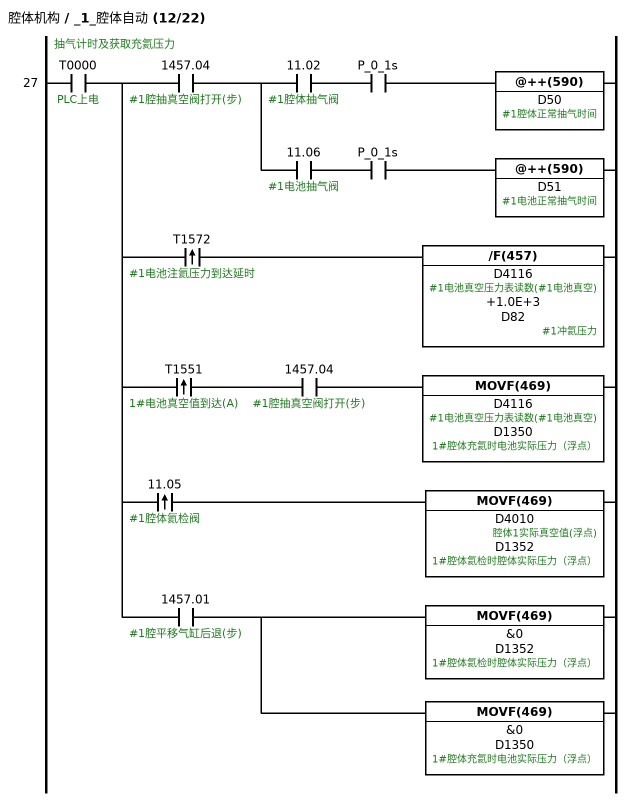
; [picture p288: 腔体机构 / _1_腔体自动, rungs 27-27]
; rung 27: 抽气计时及获取充氦压力
LD T0000  ; PLC上电
OUT TR0
AND 1457.04  ; #1腔抽真空阀打开(步)
OUT TR1
AND 11.02  ; #1腔体抽气阀
AND P_0_1s
@++(590) D50  ; #1腔体正常抽气时间
LD TR1
AND 11.06  ; #1电池抽气阀
AND P_0_1s
@++(590) D51  ; #1电池正常抽气时间
LD TR0
@AND T1572  ; #1电池注氦压力到达延时
/F(457) D4116 +1.0E+3 D82  ; #1电池真空压力表读数(#1电池真空), #1冲氦压力
LD TR0
@AND T1551  ; 1#电池真空值到达(A)
AND 1457.04  ; #1腔抽真空阀打开(步)
MOVF(469) D4116 D1350  ; #1电池真空压力表读数(#1电池真空), 1#腔体充氦时电池实际压力（浮点）
LD TR0
@AND 11.05  ; #1腔体氦检阀
MOVF(469) D4010 D1352  ; 腔体1实际真空值(浮点), 1#腔体氦检时腔体实际压力（浮点）
LD TR0
AND 1457.01  ; #1腔平移气缸后退(步)
MOVF(469) &0 D1352  ; 1#腔体氦检时腔体实际压力（浮点）
MOVF(469) &0 D1350  ; 1#腔体充氦时电池实际压力（浮点）

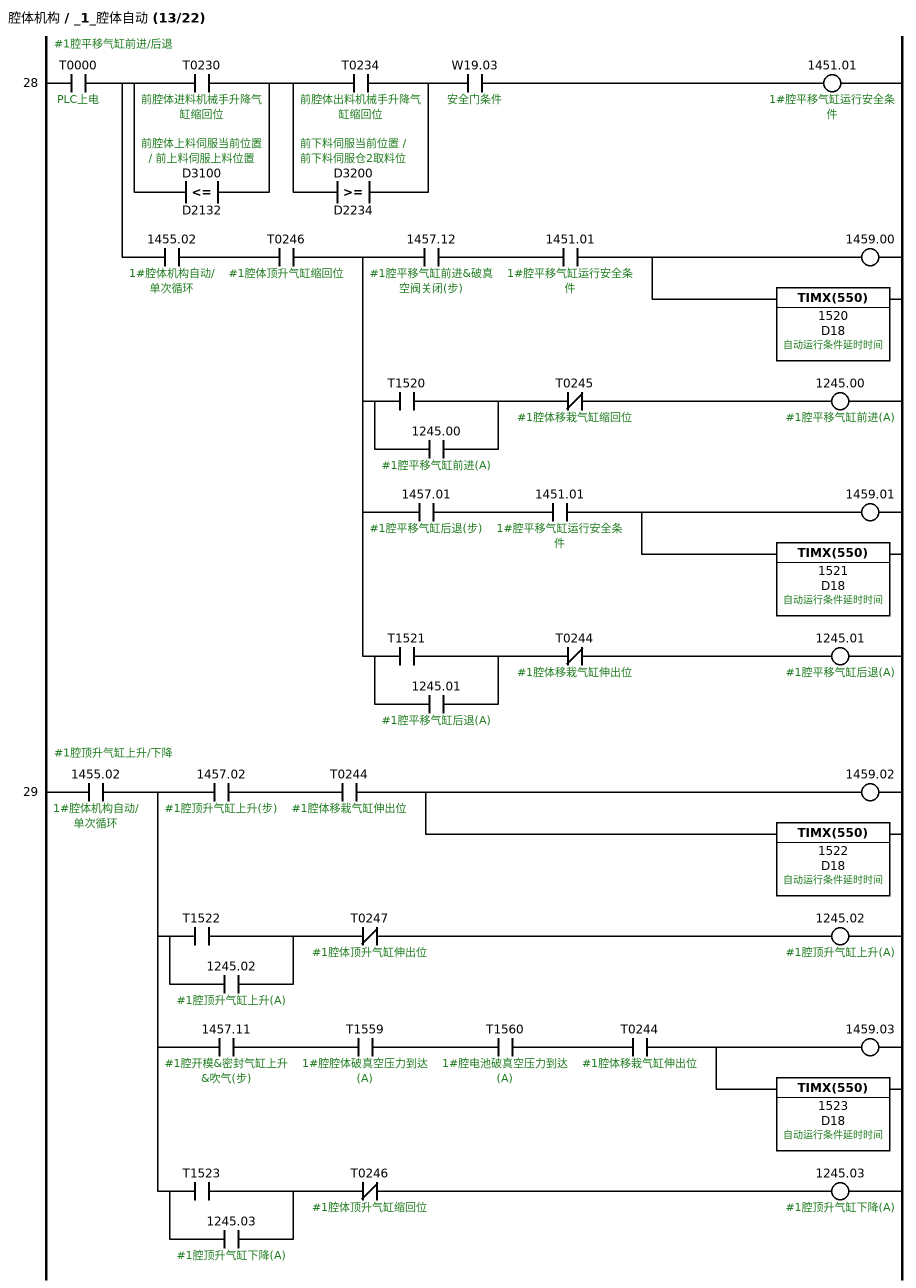
; rung 28: #1腔平移气缸前进/后退
LD T0000  ; PLC上电
OUT TR0
LD T0230  ; 前腔体进料机械手升降气缸缩回位
OR<=SL(318) D3100 D2132  ; 前腔体上料伺服当前位置, 前上料伺服上料位置
ANDLD
LD T0234  ; 前腔体出料机械手升降气缸缩回位
OR>=SL(328) D3200 D2234  ; 前下料伺服当前位置, 前下料伺服仓2取料位
ANDLD
AND W19.03  ; 安全门条件
OUT 1451.01  ; 1#腔平移气缸运行安全条件
LD TR0
AND 1455.02  ; 1#腔体机构自动/单次循环
AND T0246  ; #1腔体顶升气缸缩回位
OUT TR0
AND 1457.12  ; #1腔平移气缸前进&破真空阀关闭(步)
AND 1451.01  ; 1#腔平移气缸运行安全条件
OUT 1459.00
TIMX(550) 1520 D18  ; 自动运行条件延时时间
LD TR0
LD T1520
OR 1245.00  ; #1腔平移气缸前进(A)
ANDLD
ANDNOT T0245  ; #1腔体移栽气缸缩回位
OUT 1245.00  ; #1腔平移气缸前进(A)
LD TR0
AND 1457.01  ; #1腔平移气缸后退(步)
AND 1451.01  ; 1#腔平移气缸运行安全条件
OUT 1459.01
TIMX(550) 1521 D18  ; 自动运行条件延时时间
LD TR0
LD T1521
OR 1245.01  ; #1腔平移气缸后退(A)
ANDLD
ANDNOT T0244  ; #1腔体移栽气缸伸出位
OUT 1245.01  ; #1腔平移气缸后退(A)
; rung 29: #1腔顶升气缸上升/下降
LD 1455.02  ; 1#腔体机构自动/单次循环
OUT TR0
AND 1457.02  ; #1腔顶升气缸上升(步)
AND T0244  ; #1腔体移栽气缸伸出位
OUT 1459.02
TIMX(550) 1522 D18  ; 自动运行条件延时时间
LD TR0
LD T1522
OR 1245.02  ; #1腔顶升气缸上升(A)
ANDLD
ANDNOT T0247  ; #1腔体顶升气缸伸出位
OUT 1245.02  ; #1腔顶升气缸上升(A)
LD TR0
AND 1457.11  ; #1腔开模&密封气缸上升&吹气(步)
AND T1559  ; 1#腔腔体破真空压力到达(A)
AND T1560  ; 1#腔电池破真空压力到达(A)
AND T0244  ; #1腔体移栽气缸伸出位
OUT 1459.03
TIMX(550) 1523 D18  ; 自动运行条件延时时间
LD TR0
LD T1523
OR 1245.03  ; #1腔顶升气缸下降(A)
ANDLD
ANDNOT T0246  ; #1腔体顶升气缸缩回位
OUT 1245.03  ; #1腔顶升气缸下降(A)

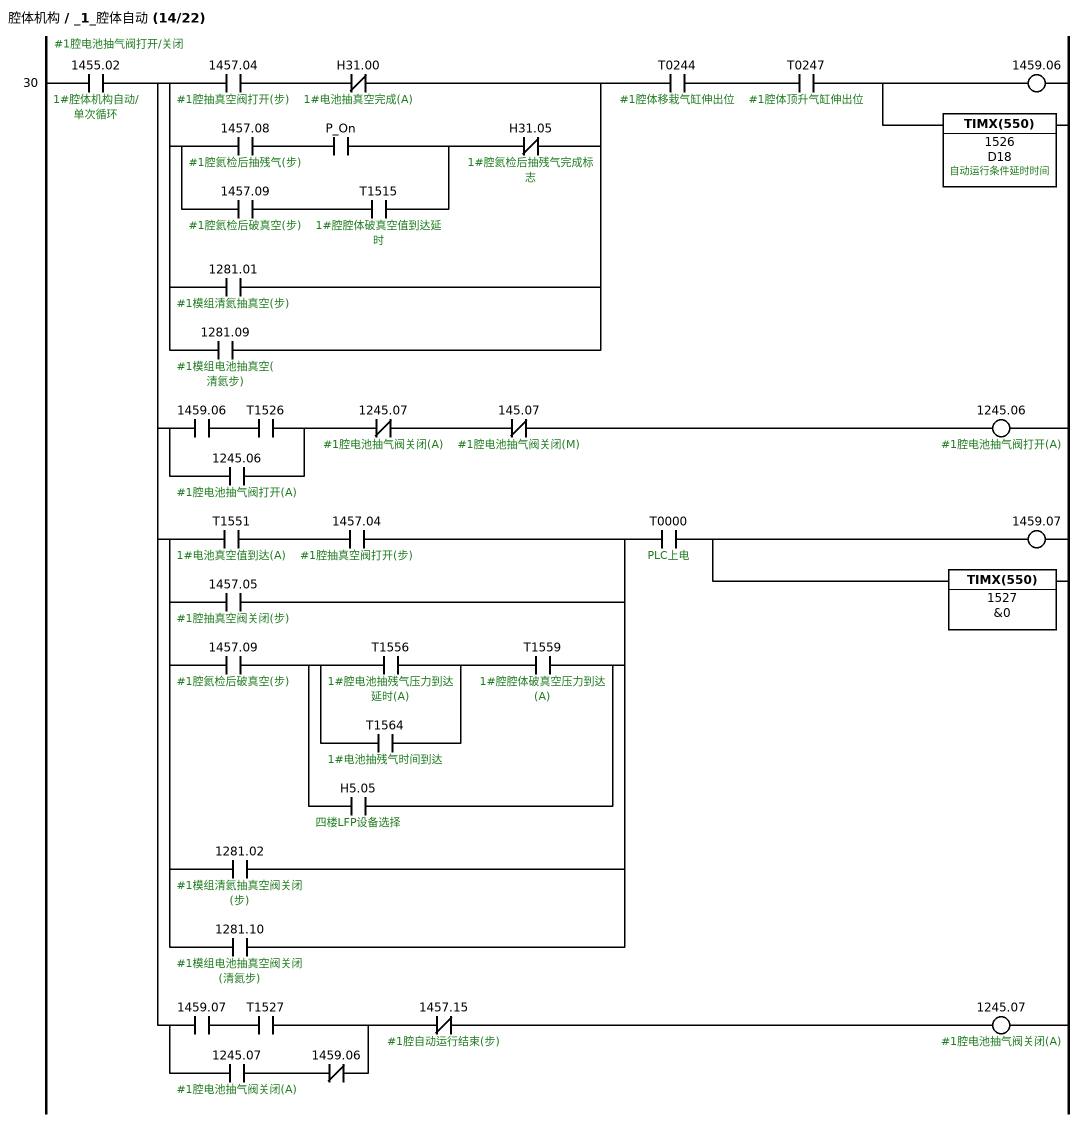
; rung 30: #1腔电池抽气阀打开/关闭
LD 1455.02  ; 1#腔体机构自动/单次循环
OUT TR0
LD 1457.04  ; #1腔抽真空阀打开(步)
ANDNOT H31.00  ; 1#电池抽真空完成(A)
LD 1457.08  ; #1腔氦检后抽残气(步)
AND P_On
LD 1457.09  ; #1腔氦检后破真空(步)
AND T1515  ; 1#腔腔体破真空值到达延时
ORLD
ANDNOT H31.05  ; 1#腔氦检后抽残气完成标志
ORLD
OR 1281.01  ; #1模组清氦抽真空(步)
OR 1281.09  ; #1模组电池抽真空(清氦步)
ANDLD
AND T0244  ; #1腔体移栽气缸伸出位
AND T0247  ; #1腔体顶升气缸伸出位
OUT 1459.06
TIMX(550) 1526 D18  ; 自动运行条件延时时间
LD TR0
LD 1459.06
AND T1526
OR 1245.06  ; #1腔电池抽气阀打开(A)
ANDLD
ANDNOT 1245.07  ; #1腔电池抽气阀关闭(A)
ANDNOT 145.07  ; #1腔电池抽气阀关闭(M)
OUT 1245.06  ; #1腔电池抽气阀打开(A)
LD TR0
LD T1551  ; 1#电池真空值到达(A)
AND 1457.04  ; #1腔抽真空阀打开(步)
OR 1457.05  ; #1腔抽真空阀关闭(步)
LD 1457.09  ; #1腔氦检后破真空(步)
LD T1556  ; 1#腔电池抽残气压力到达延时(A)
OR T1564  ; 1#电池抽残气时间到达
AND T1559  ; 1#腔腔体破真空压力到达(A)
OR H5.05  ; 四楼LFP设备选择
ANDLD
ORLD
OR 1281.02  ; #1模组清氦抽真空阀关闭(步)
OR 1281.10  ; #1模组电池抽真空阀关闭(清氦步)
ANDLD
AND T0000  ; PLC上电
OUT 1459.07
TIMX(550) 1527 &0
LD TR0
LD 1459.07
AND T1527
LD 1245.07  ; #1腔电池抽气阀关闭(A)
ANDNOT 1459.06
ORLD
ANDLD
ANDNOT 1457.15  ; #1腔自动运行结束(步)
OUT 1245.07  ; #1腔电池抽气阀关闭(A)

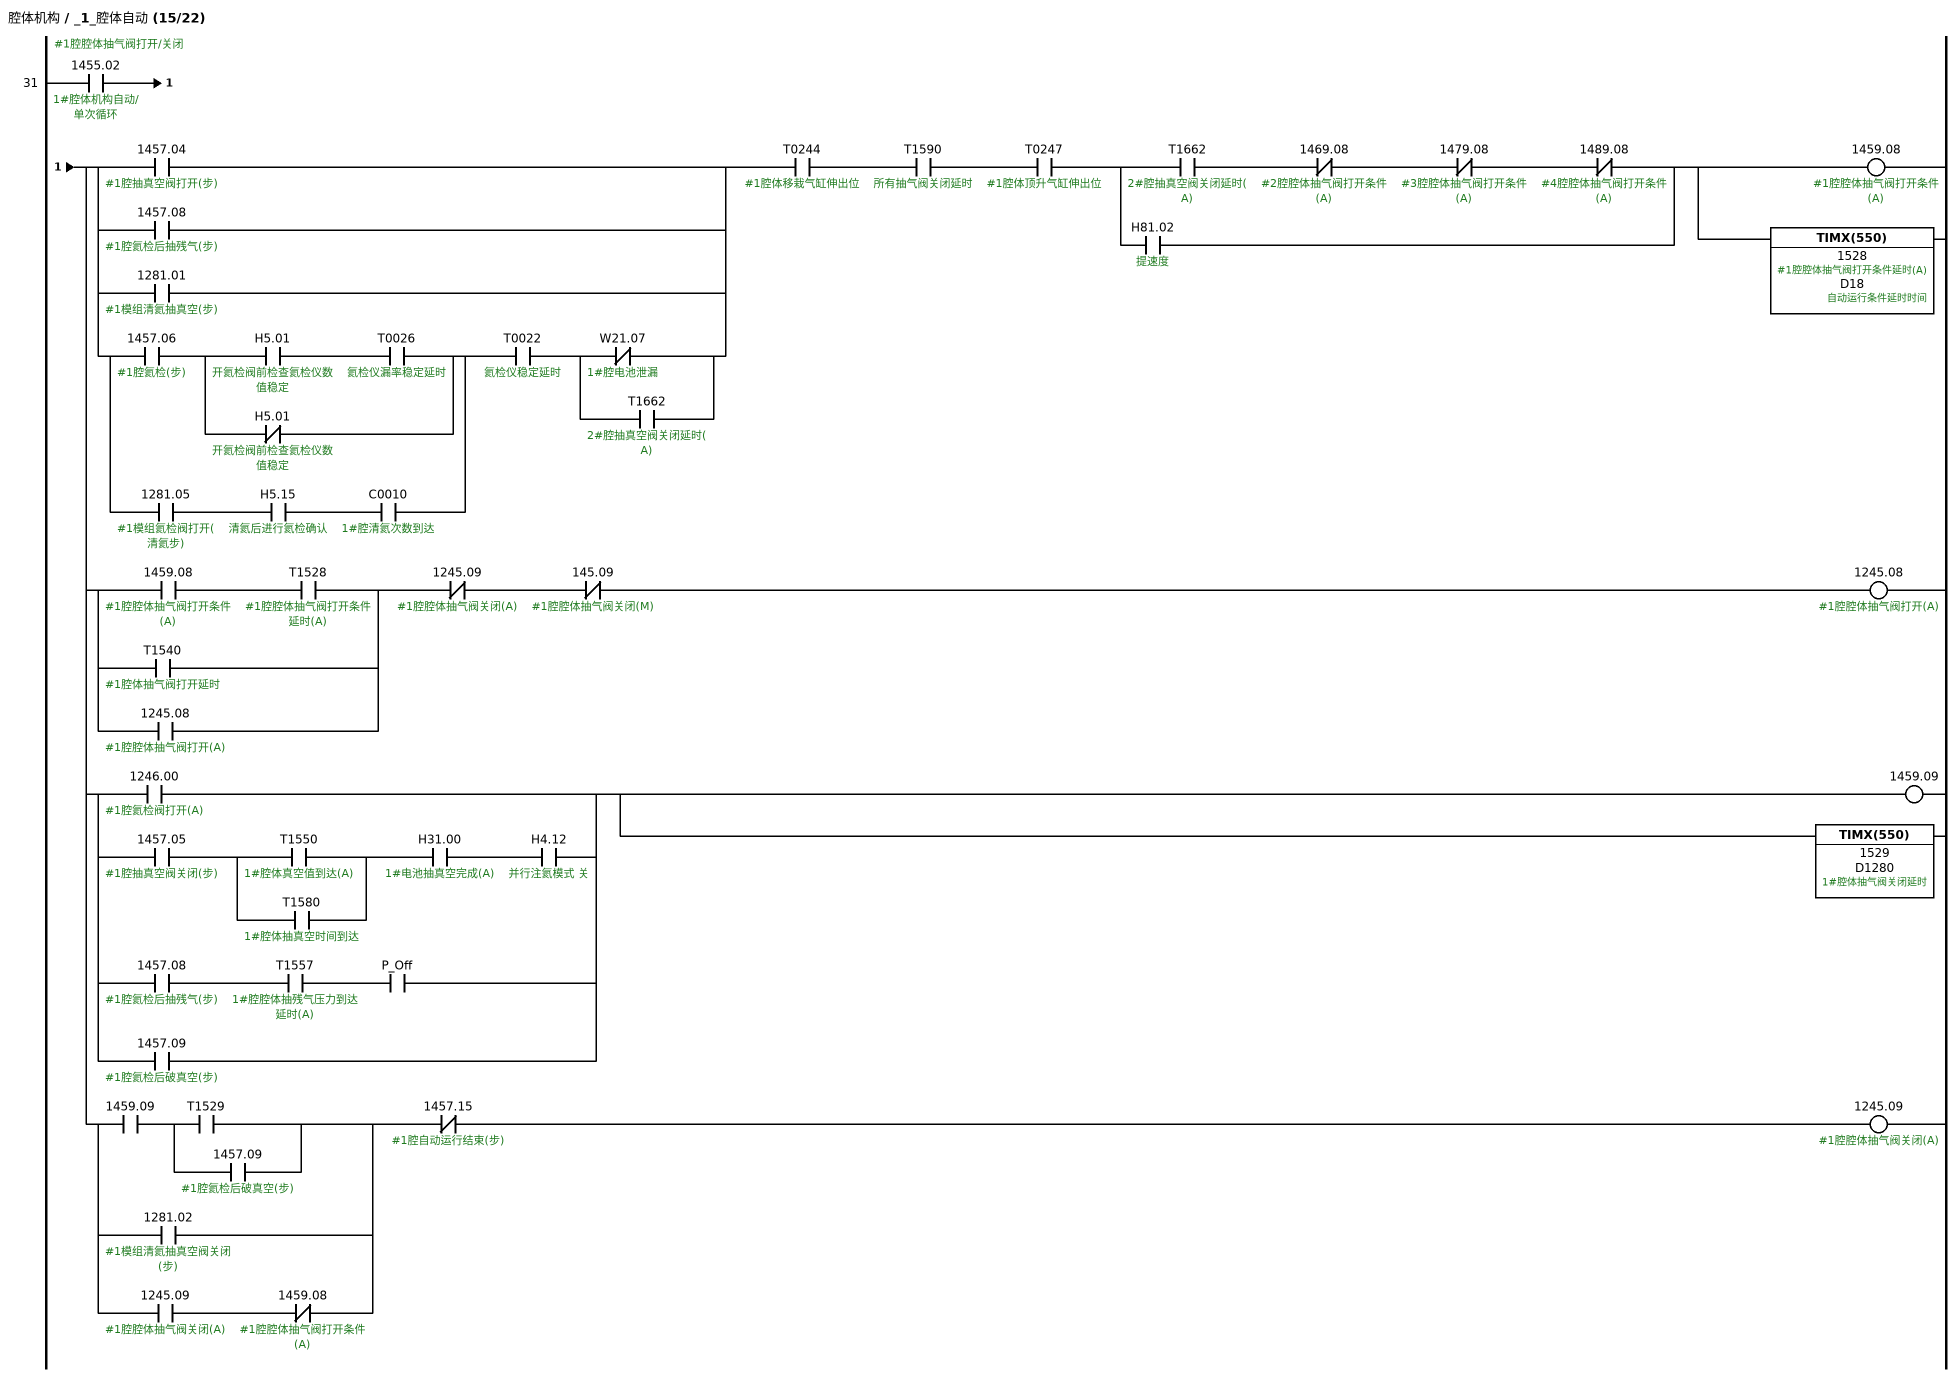
; rung 31: #1腔腔体抽气阀打开/关闭
LD 1455.02  ; 1#腔体机构自动/单次循环
OUT TR0
LD 1457.04  ; #1腔抽真空阀打开(步)
OR 1457.08  ; #1腔氦检后抽残气(步)
OR 1281.01  ; #1模组清氦抽真空(步)
LD 1457.06  ; #1腔氦检(步)
LD H5.01  ; 开氦检阀前检查氦检仪数值稳定
AND T0026  ; 氦检仪漏率稳定延时
ORNOT H5.01  ; 开氦检阀前检查氦检仪数值稳定
ANDLD
LD 1281.05  ; #1模组氦检阀打开(清氦步)
AND H5.15  ; 清氦后进行氦检确认
AND C0010  ; 1#腔清氦次数到达
ORLD
AND T0022  ; 氦检仪稳定延时
LDNOT W21.07  ; 1#腔电池泄漏
OR T1662  ; 2#腔抽真空阀关闭延时(A)
ANDLD
ORLD
ANDLD
AND T0244  ; #1腔体移栽气缸伸出位
AND T1590  ; 所有抽气阀关闭延时
AND T0247  ; #1腔体顶升气缸伸出位
LD T1662  ; 2#腔抽真空阀关闭延时(A)
ANDNOT 1469.08  ; #2腔腔体抽气阀打开条件(A)
ANDNOT 1479.08  ; #3腔腔体抽气阀打开条件(A)
ANDNOT 1489.08  ; #4腔腔体抽气阀打开条件(A)
OR H81.02  ; 提速度
ANDLD
OUT 1459.08  ; #1腔腔体抽气阀打开条件(A)
TIMX(550) 1528 D18  ; 自动运行条件延时时间, #1腔腔体抽气阀打开条件延时(A)
LD TR0
LD 1459.08  ; #1腔腔体抽气阀打开条件(A)
AND T1528  ; #1腔腔体抽气阀打开条件延时(A)
OR T1540  ; #1腔体抽气阀打开延时
OR 1245.08  ; #1腔腔体抽气阀打开(A)
ANDLD
ANDNOT 1245.09  ; #1腔腔体抽气阀关闭(A)
ANDNOT 145.09  ; #1腔腔体抽气阀关闭(M)
OUT 1245.08  ; #1腔腔体抽气阀打开(A)
LD TR0
LD 1246.00  ; #1腔氦检阀打开(A)
LD 1457.05  ; #1腔抽真空阀关闭(步)
LD T1550  ; 1#腔体真空值到达(A)
OR T1580  ; 1#腔体抽真空时间到达
ANDLD
AND H31.00  ; 1#电池抽真空完成(A)
AND H4.12  ; 并行注氦模式 关
ORLD
LD 1457.08  ; #1腔氦检后抽残气(步)
AND T1557  ; 1#腔腔体抽残气压力到达延时(A)
AND P_Off
ORLD
OR 1457.09  ; #1腔氦检后破真空(步)
ANDLD
OUT 1459.09
TIMX(550) 1529 D1280  ; 1#腔体抽气阀关闭延时
LD TR0
LD 1459.09
LD T1529
OR 1457.09  ; #1腔氦检后破真空(步)
ANDLD
OR 1281.02  ; #1模组清氦抽真空阀关闭(步)
LD 1245.09  ; #1腔腔体抽气阀关闭(A)
ANDNOT 1459.08  ; #1腔腔体抽气阀打开条件(A)
ORLD
ANDLD
ANDNOT 1457.15  ; #1腔自动运行结束(步)
OUT 1245.09  ; #1腔腔体抽气阀关闭(A)

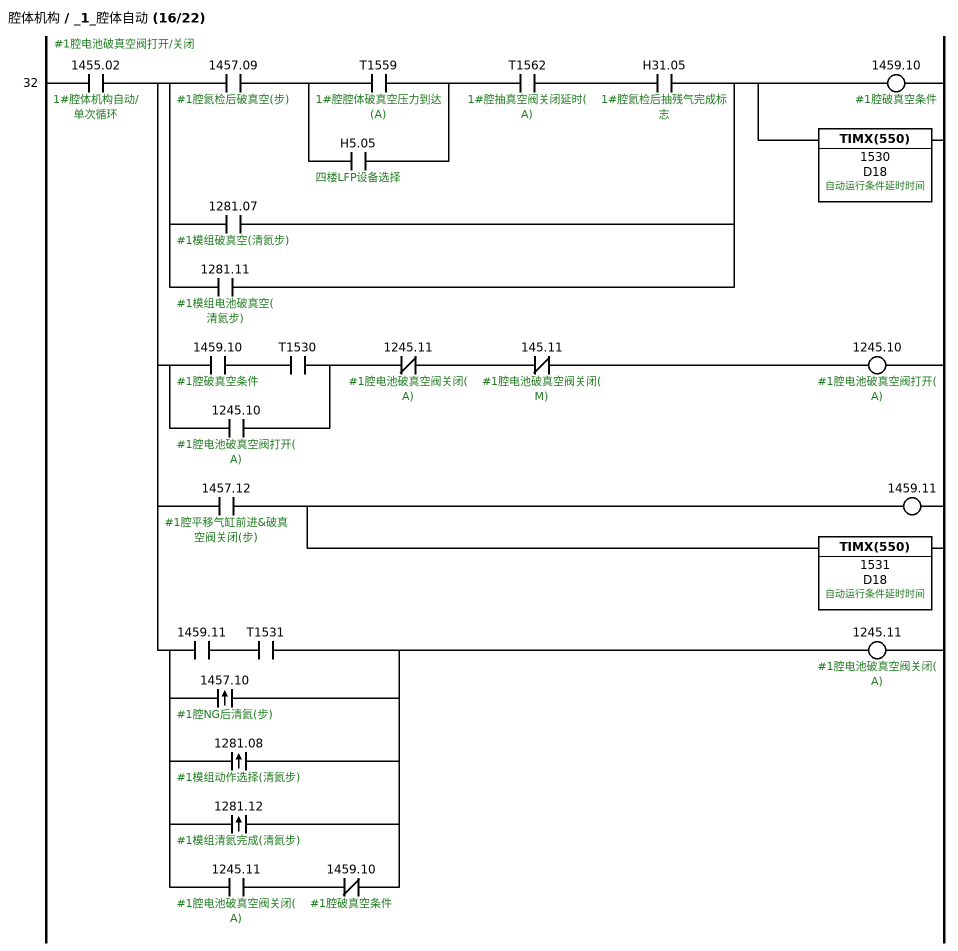
; rung 32: #1腔电池破真空阀打开/关闭
LD 1455.02  ; 1#腔体机构自动/单次循环
OUT TR0
LD 1457.09  ; #1腔氦检后破真空(步)
LD T1559  ; 1#腔腔体破真空压力到达(A)
OR H5.05  ; 四楼LFP设备选择
ANDLD
AND T1562  ; 1#腔抽真空阀关闭延时(A)
AND H31.05  ; 1#腔氦检后抽残气完成标志
OR 1281.07  ; #1模组破真空(清氦步)
OR 1281.11  ; #1模组电池破真空(清氦步)
ANDLD
OUT 1459.10  ; #1腔破真空条件
TIMX(550) 1530 D18  ; 自动运行条件延时时间
LD TR0
LD 1459.10  ; #1腔破真空条件
AND T1530
OR 1245.10  ; #1腔电池破真空阀打开(A)
ANDLD
ANDNOT 1245.11  ; #1腔电池破真空阀关闭(A)
ANDNOT 145.11  ; #1腔电池破真空阀关闭(M)
OUT 1245.10  ; #1腔电池破真空阀打开(A)
LD TR0
AND 1457.12  ; #1腔平移气缸前进&破真空阀关闭(步)
OUT 1459.11
TIMX(550) 1531 D18  ; 自动运行条件延时时间
LD TR0
LD 1459.11
AND T1531
@OR 1457.10  ; #1腔NG后清氦(步)
@OR 1281.08  ; #1模组动作选择(清氦步)
@OR 1281.12  ; #1模组清氦完成(清氦步)
LD 1245.11  ; #1腔电池破真空阀关闭(A)
ANDNOT 1459.10  ; #1腔破真空条件
ORLD
ANDLD
OUT 1245.11  ; #1腔电池破真空阀关闭(A)

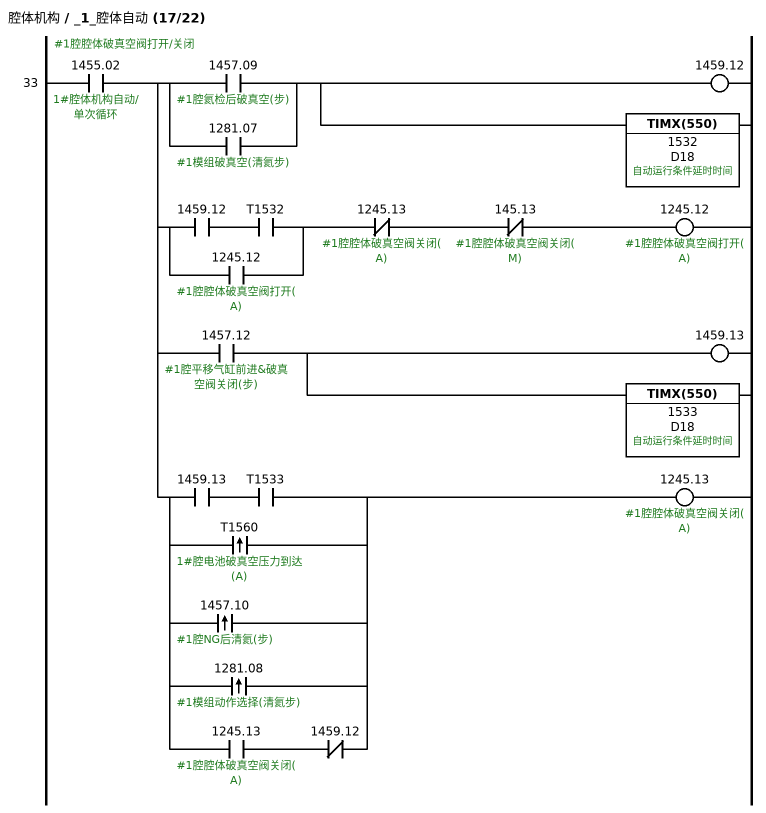
; rung 33: #1腔腔体破真空阀打开/关闭
LD 1455.02  ; 1#腔体机构自动/单次循环
OUT TR0
LD 1457.09  ; #1腔氦检后破真空(步)
OR 1281.07  ; #1模组破真空(清氦步)
ANDLD
OUT 1459.12
TIMX(550) 1532 D18  ; 自动运行条件延时时间
LD TR0
LD 1459.12
AND T1532
OR 1245.12  ; #1腔腔体破真空阀打开(A)
ANDLD
ANDNOT 1245.13  ; #1腔腔体破真空阀关闭(A)
ANDNOT 145.13  ; #1腔腔体破真空阀关闭(M)
OUT 1245.12  ; #1腔腔体破真空阀打开(A)
LD TR0
AND 1457.12  ; #1腔平移气缸前进&破真空阀关闭(步)
OUT 1459.13
TIMX(550) 1533 D18  ; 自动运行条件延时时间
LD TR0
LD 1459.13
AND T1533
@OR T1560  ; 1#腔电池破真空压力到达(A)
@OR 1457.10  ; #1腔NG后清氦(步)
@OR 1281.08  ; #1模组动作选择(清氦步)
LD 1245.13  ; #1腔腔体破真空阀关闭(A)
ANDNOT 1459.12
ORLD
ANDLD
OUT 1245.13  ; #1腔腔体破真空阀关闭(A)

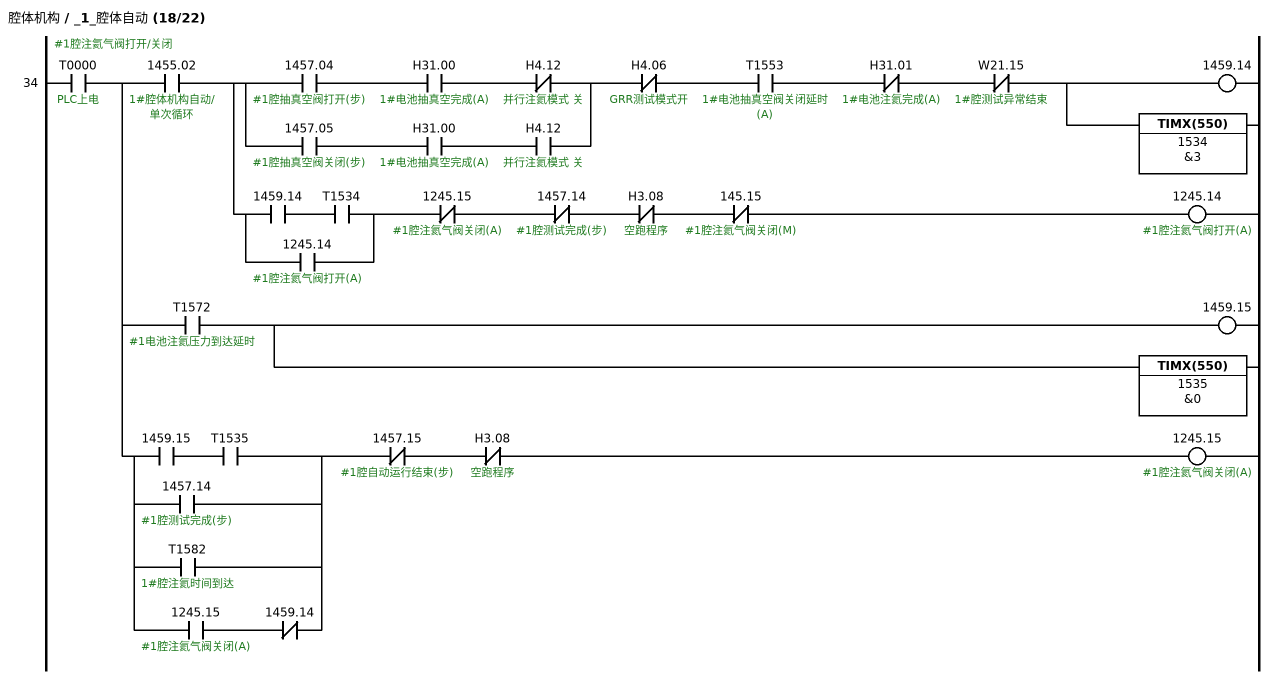
; rung 34: #1腔注氦气阀打开/关闭
LD T0000  ; PLC上电
OUT TR0
AND 1455.02  ; 1#腔体机构自动/单次循环
OUT TR1
LD 1457.04  ; #1腔抽真空阀打开(步)
AND H31.00  ; 1#电池抽真空完成(A)
ANDNOT H4.12  ; 并行注氦模式 关
LD 1457.05  ; #1腔抽真空阀关闭(步)
AND H31.00  ; 1#电池抽真空完成(A)
AND H4.12  ; 并行注氦模式 关
ORLD
ANDLD
ANDNOT H4.06  ; GRR测试模式开
AND T1553  ; 1#电池抽真空阀关闭延时(A)
ANDNOT H31.01  ; 1#电池注氦完成(A)
ANDNOT W21.15  ; 1#腔测试异常结束
OUT 1459.14
TIMX(550) 1534 &3
LD TR1
LD 1459.14
AND T1534
OR 1245.14  ; #1腔注氦气阀打开(A)
ANDLD
ANDNOT 1245.15  ; #1腔注氦气阀关闭(A)
ANDNOT 1457.14  ; #1腔测试完成(步)
ANDNOT H3.08  ; 空跑程序
ANDNOT 145.15  ; #1腔注氦气阀关闭(M)
OUT 1245.14  ; #1腔注氦气阀打开(A)
LD TR0
AND T1572  ; #1电池注氦压力到达延时
OUT 1459.15
TIMX(550) 1535 &0
LD TR0
LD 1459.15
AND T1535
OR 1457.14  ; #1腔测试完成(步)
OR T1582  ; 1#腔注氦时间到达
LD 1245.15  ; #1腔注氦气阀关闭(A)
ANDNOT 1459.14
ORLD
ANDLD
ANDNOT 1457.15  ; #1腔自动运行结束(步)
ANDNOT H3.08  ; 空跑程序
OUT 1245.15  ; #1腔注氦气阀关闭(A)

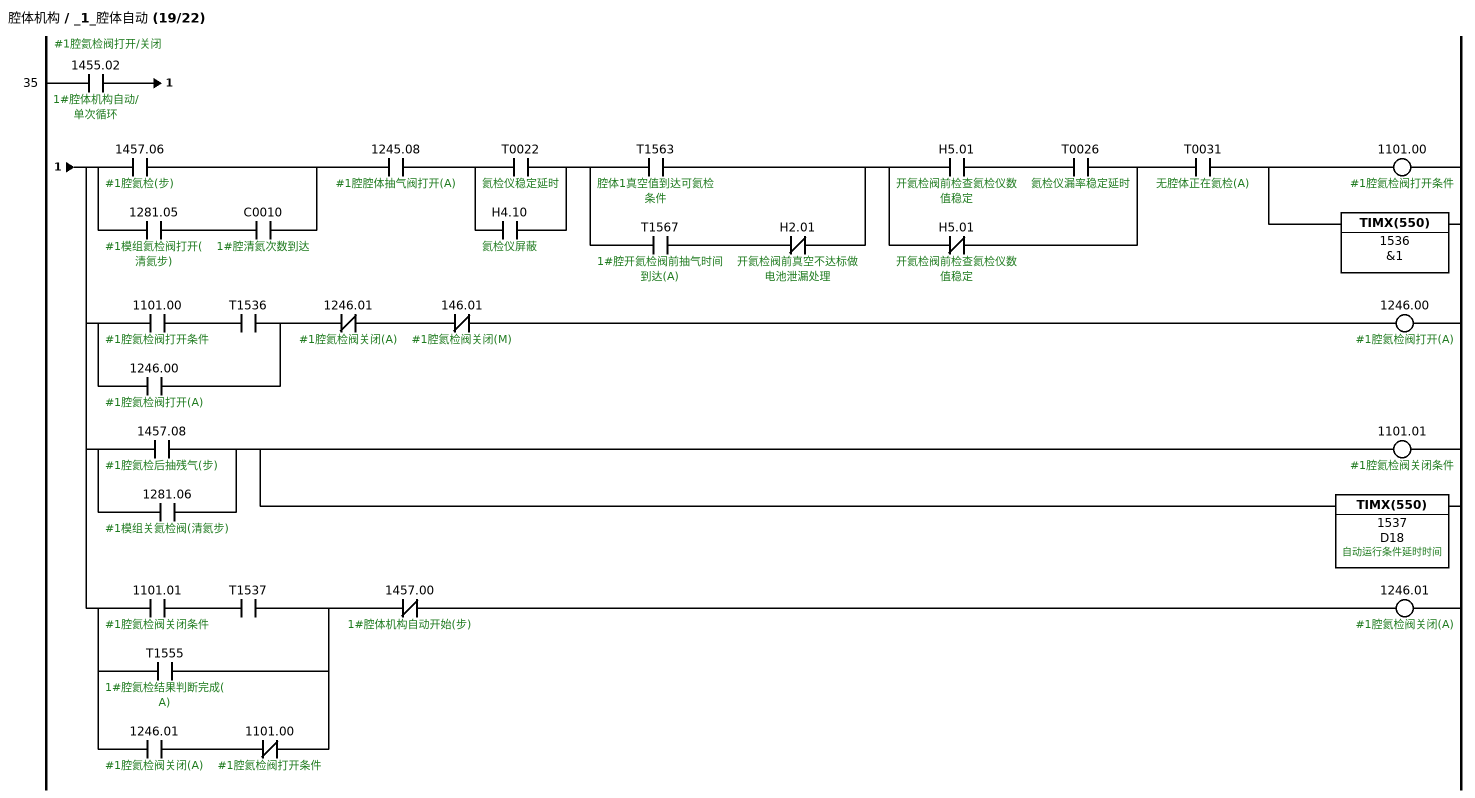
; rung 35: #1腔氦检阀打开/关闭
LD 1455.02  ; 1#腔体机构自动/单次循环
OUT TR0
LD 1457.06  ; #1腔氦检(步)
LD 1281.05  ; #1模组氦检阀打开(清氦步)
AND C0010  ; 1#腔清氦次数到达
ORLD
ANDLD
AND 1245.08  ; #1腔腔体抽气阀打开(A)
LD T0022  ; 氦检仪稳定延时
OR H4.10  ; 氦检仪屏蔽
ANDLD
LD T1563  ; 腔体1真空值到达可氦检条件
LD T1567  ; 1#腔开氦检阀前抽气时间到达(A)
ANDNOT H2.01  ; 开氦检阀前真空不达标做电池泄漏处理
ORLD
ANDLD
LD H5.01  ; 开氦检阀前检查氦检仪数值稳定
AND T0026  ; 氦检仪漏率稳定延时
ORNOT H5.01  ; 开氦检阀前检查氦检仪数值稳定
ANDLD
AND T0031  ; 无腔体正在氦检(A)
OUT 1101.00  ; #1腔氦检阀打开条件
TIMX(550) 1536 &1
LD TR0
LD 1101.00  ; #1腔氦检阀打开条件
AND T1536
OR 1246.00  ; #1腔氦检阀打开(A)
ANDLD
ANDNOT 1246.01  ; #1腔氦检阀关闭(A)
ANDNOT 146.01  ; #1腔氦检阀关闭(M)
OUT 1246.00  ; #1腔氦检阀打开(A)
LD TR0
LD 1457.08  ; #1腔氦检后抽残气(步)
OR 1281.06  ; #1模组关氦检阀(清氦步)
ANDLD
OUT 1101.01  ; #1腔氦检阀关闭条件
TIMX(550) 1537 D18  ; 自动运行条件延时时间
LD TR0
LD 1101.01  ; #1腔氦检阀关闭条件
AND T1537
OR T1555  ; 1#腔氦检结果判断完成(A)
LD 1246.01  ; #1腔氦检阀关闭(A)
ANDNOT 1101.00  ; #1腔氦检阀打开条件
ORLD
ANDLD
ANDNOT 1457.00  ; 1#腔体机构自动开始(步)
OUT 1246.01  ; #1腔氦检阀关闭(A)

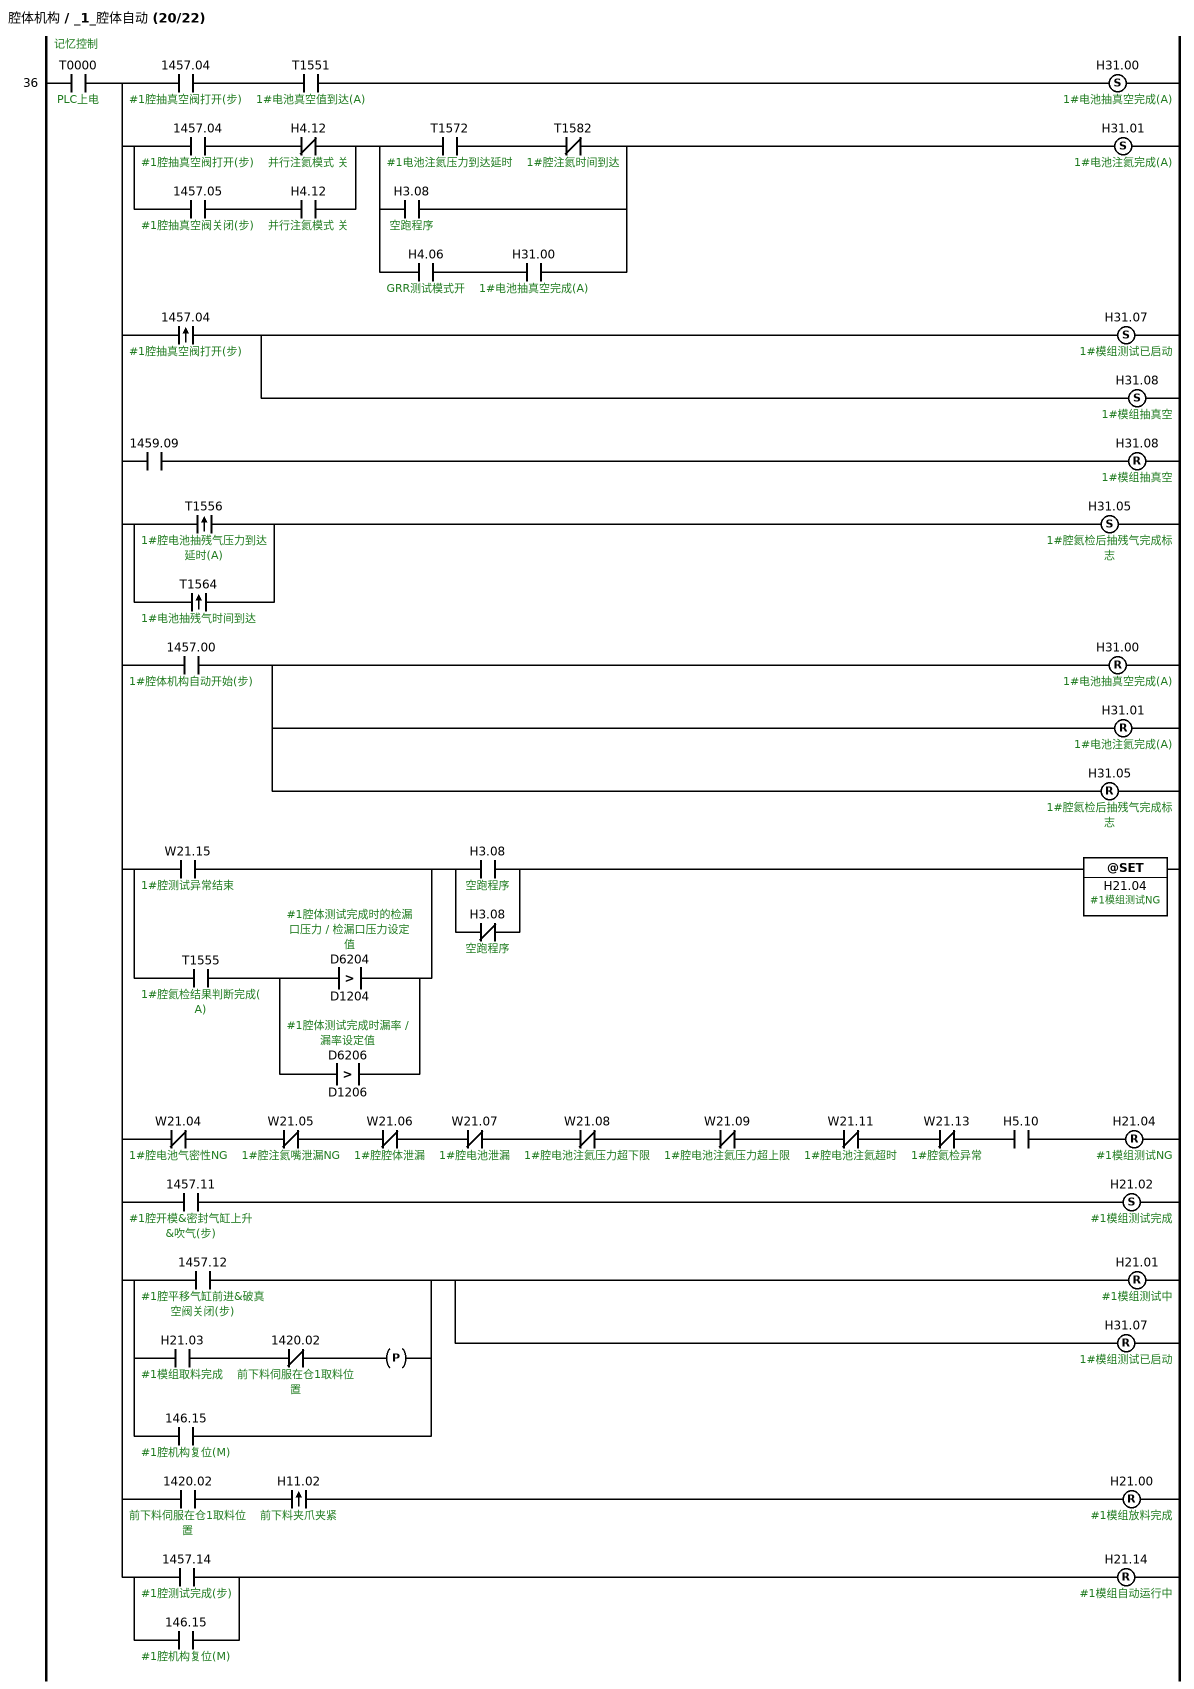
; rung 36: 记忆控制
LD T0000  ; PLC上电
OUT TR0
AND 1457.04  ; #1腔抽真空阀打开(步)
AND T1551  ; 1#电池真空值到达(A)
SET H31.00  ; 1#电池抽真空完成(A)
LD TR0
LD 1457.04  ; #1腔抽真空阀打开(步)
ANDNOT H4.12  ; 并行注氦模式 关
LD 1457.05  ; #1腔抽真空阀关闭(步)
AND H4.12  ; 并行注氦模式 关
ORLD
ANDLD
LD T1572  ; #1电池注氦压力到达延时
ANDNOT T1582  ; 1#腔注氦时间到达
OR H3.08  ; 空跑程序
LD H4.06  ; GRR测试模式开
AND H31.00  ; 1#电池抽真空完成(A)
ORLD
ANDLD
SET H31.01  ; 1#电池注氦完成(A)
LD TR0
@AND 1457.04  ; #1腔抽真空阀打开(步)
SET H31.07  ; 1#模组测试已启动
SET H31.08  ; 1#模组抽真空
LD TR0
AND 1459.09
RSET H31.08  ; 1#模组抽真空
LD TR0
@LD T1556  ; 1#腔电池抽残气压力到达延时(A)
@OR T1564  ; 1#电池抽残气时间到达
ANDLD
SET H31.05  ; 1#腔氦检后抽残气完成标志
LD TR0
AND 1457.00  ; 1#腔体机构自动开始(步)
RSET H31.00  ; 1#电池抽真空完成(A)
RSET H31.01  ; 1#电池注氦完成(A)
RSET H31.05  ; 1#腔氦检后抽残气完成标志
LD TR0
LD W21.15  ; 1#腔测试异常结束
LD T1555  ; 1#腔氦检结果判断完成(A)
LD>F(333) D6204 D1204  ; #1腔体测试完成时的检漏口压力, 检漏口压力设定值
OR>F(333) D6206 D1206  ; #1腔体测试完成时漏率, 漏率设定值
ANDLD
ORLD
ANDLD
LD H3.08  ; 空跑程序
ORNOT H3.08  ; 空跑程序
ANDLD
@SET H21.04  ; #1模组测试NG
LD TR0
ANDNOT W21.04  ; 1#腔电池气密性NG
ANDNOT W21.05  ; 1#腔注氦嘴泄漏NG
ANDNOT W21.06  ; 1#腔腔体泄漏
ANDNOT W21.07  ; 1#腔电池泄漏
ANDNOT W21.08  ; 1#腔电池注氦压力超下限
ANDNOT W21.09  ; 1#腔电池注氦压力超上限
ANDNOT W21.11  ; 1#腔电池注氦超时
ANDNOT W21.13  ; 1#腔氦检异常
AND H5.10
RSET H21.04  ; #1模组测试NG
LD TR0
AND 1457.11  ; #1腔开模&密封气缸上升&吹气(步)
SET H21.02  ; #1模组测试完成
LD TR0
LD 1457.12  ; #1腔平移气缸前进&破真空阀关闭(步)
LD H21.03  ; #1模组取料完成
ANDNOT 1420.02  ; 前下料伺服在仓1取料位置
UP(521)
ORLD
OR 146.15  ; #1腔机构复位(M)
ANDLD
RSET H21.01  ; #1模组测试中
RSET H31.07  ; 1#模组测试已启动
LD TR0
AND 1420.02  ; 前下料伺服在仓1取料位置
@AND H11.02  ; 前下料夹爪夹紧
RSET H21.00  ; #1模组放料完成
LD TR0
LD 1457.14  ; #1腔测试完成(步)
OR 146.15  ; #1腔机构复位(M)
ANDLD
RSET H21.14  ; #1模组自动运行中

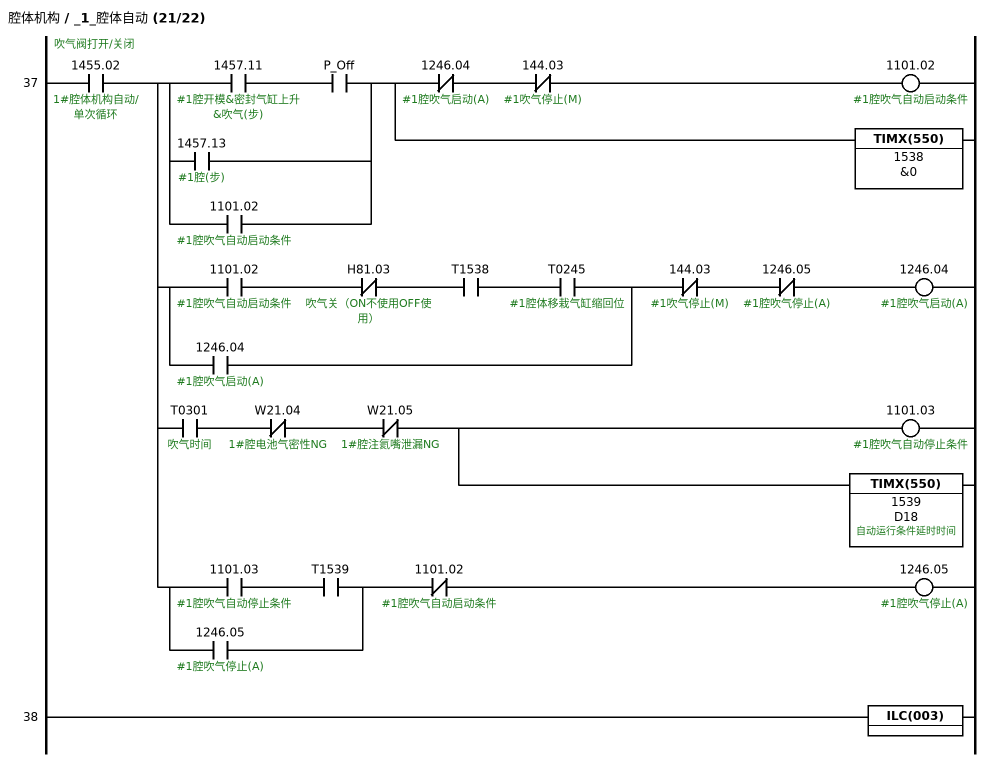
; rung 37: 吹气阀打开/关闭
LD 1455.02  ; 1#腔体机构自动/单次循环
OUT TR0
LD 1457.11  ; #1腔开模&密封气缸上升&吹气(步)
AND P_Off
OR 1457.13  ; #1腔(步)
OR 1101.02  ; #1腔吹气自动启动条件
ANDLD
OUT TR1
ANDNOT 1246.04  ; #1腔吹气启动(A)
ANDNOT 144.03  ; #1吹气停止(M)
OUT 1101.02  ; #1腔吹气自动启动条件
LD TR1
TIMX(550) 1538 &0
LD TR0
LD 1101.02  ; #1腔吹气自动启动条件
ANDNOT H81.03  ; 吹气关（ON不使用OFF使用）
AND T1538
AND T0245  ; #1腔体移栽气缸缩回位
OR 1246.04  ; #1腔吹气启动(A)
ANDLD
ANDNOT 144.03  ; #1吹气停止(M)
ANDNOT 1246.05  ; #1腔吹气停止(A)
OUT 1246.04  ; #1腔吹气启动(A)
LD TR0
AND T0301  ; 吹气时间
ANDNOT W21.04  ; 1#腔电池气密性NG
ANDNOT W21.05  ; 1#腔注氦嘴泄漏NG
OUT 1101.03  ; #1腔吹气自动停止条件
TIMX(550) 1539 D18  ; 自动运行条件延时时间
LD TR0
LD 1101.03  ; #1腔吹气自动停止条件
AND T1539
OR 1246.05  ; #1腔吹气停止(A)
ANDLD
ANDNOT 1101.02  ; #1腔吹气自动启动条件
OUT 1246.05  ; #1腔吹气停止(A)
; rung 38
ILC(003)

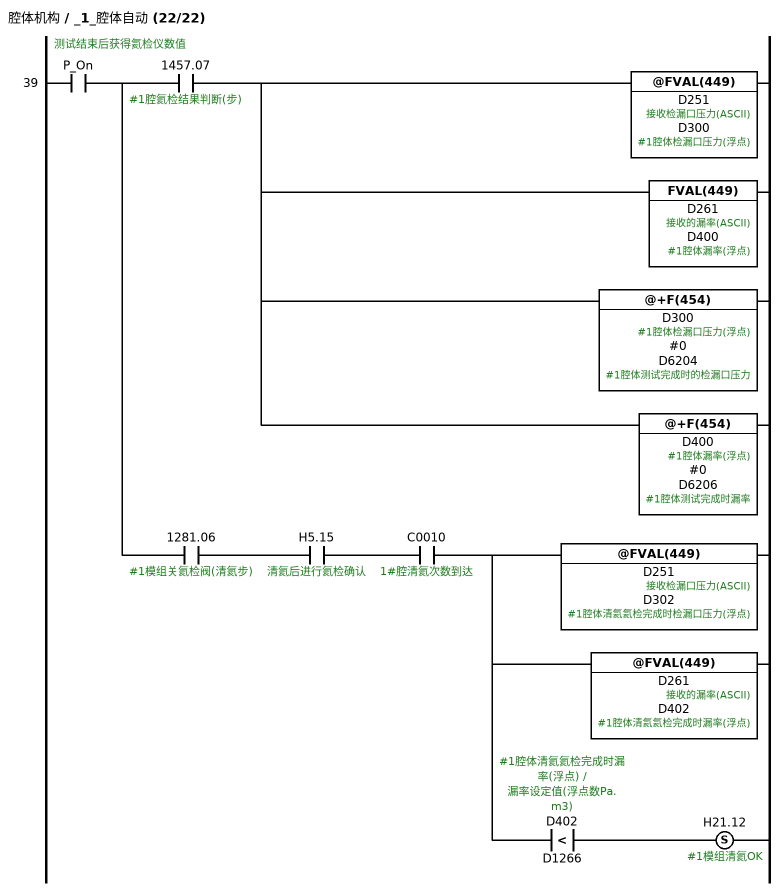
; rung 39: 测试结束后获得氦检仪数值
LD P_On
OUT TR0
AND 1457.07  ; #1腔氦检结果判断(步)
@FVAL(449) D251 D300  ; 接收检漏口压力(ASCII), #1腔体检漏口压力(浮点)
FVAL(449) D261 D400  ; 接收的漏率(ASCII), #1腔体漏率(浮点)
@+F(454) D300 #0 D6204  ; #1腔体检漏口压力(浮点), #1腔体测试完成时的检漏口压力
@+F(454) D400 #0 D6206  ; #1腔体漏率(浮点), #1腔体测试完成时漏率
LD TR0
AND 1281.06  ; #1模组关氦检阀(清氦步)
AND H5.15  ; 清氦后进行氦检确认
AND C0010  ; 1#腔清氦次数到达
@FVAL(449) D251 D302  ; 接收检漏口压力(ASCII), #1腔体清氦氦检完成时检漏口压力(浮点)
@FVAL(449) D261 D402  ; 接收的漏率(ASCII), #1腔体清氦氦检完成时漏率(浮点)
AND<F(331) D402 D1266  ; #1腔体清氦氦检完成时漏率(浮点), 漏率设定值(浮点数Pa.m3)
SET H21.12  ; #1模组清氦OK

### Section _2_腔体自动

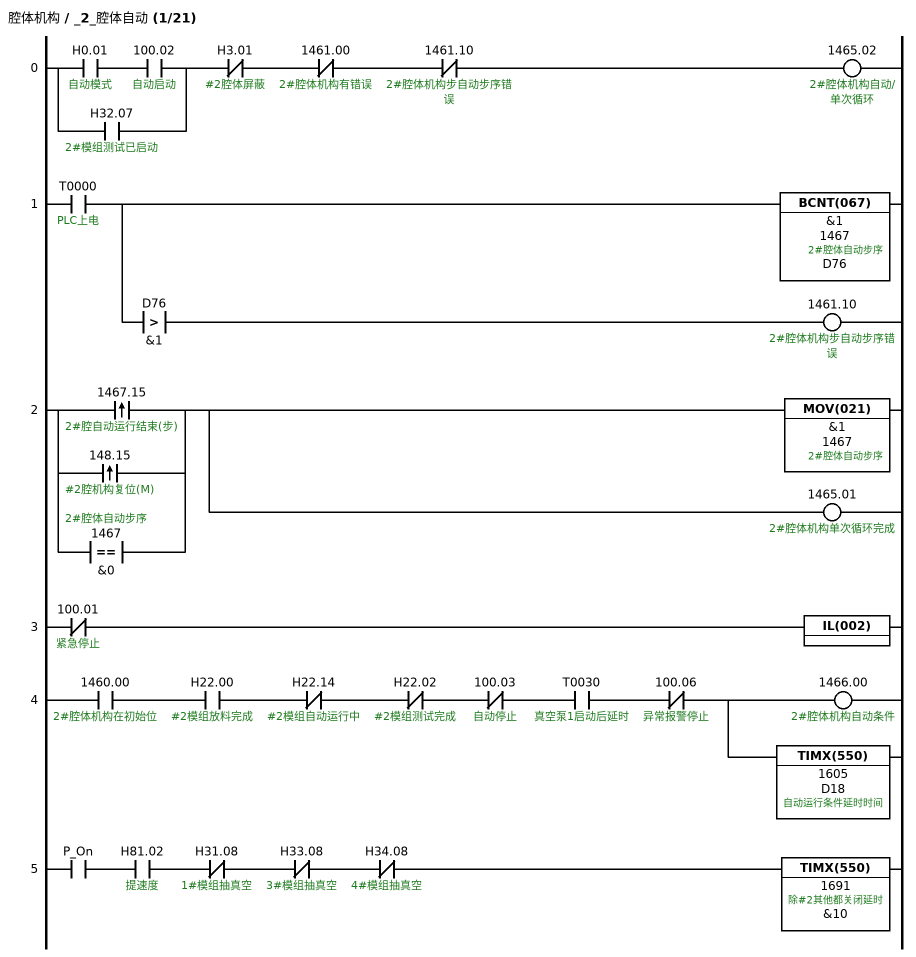
; rung 0
LD H0.01  ; 自动模式
AND 100.02  ; 自动启动
OR H32.07  ; 2#模组测试已启动
ANDNOT H3.01  ; #2腔体屏蔽
ANDNOT 1461.00  ; 2#腔体机构有错误
ANDNOT 1461.10  ; 2#腔体机构步自动步序错误
OUT 1465.02  ; 2#腔体机构自动/单次循环
; rung 1
LD T0000  ; PLC上电
BCNT(067) &1 1467 D76  ; 2#腔体自动步序
AND>(320) D76 &1
OUT 1461.10  ; 2#腔体机构步自动步序错误
; rung 2
@LD 1467.15  ; 2#腔自动运行结束(步)
@OR 148.15  ; #2腔机构复位(M)
OR=(300) 1467 &0  ; 2#腔体自动步序
MOV(021) &1 1467  ; 2#腔体自动步序
OUT 1465.01  ; 2#腔体机构单次循环完成
; rung 3
LDNOT 100.01  ; 紧急停止
IL(002)
; rung 4
LD 1460.00  ; 2#腔体机构在初始位
AND H22.00  ; #2模组放料完成
ANDNOT H22.14  ; #2模组自动运行中
ANDNOT H22.02  ; #2模组测试完成
ANDNOT 100.03  ; 自动停止
AND T0030  ; 真空泵1启动后延时
ANDNOT 100.06  ; 异常报警停止
OUT 1466.00  ; 2#腔体机构自动条件
TIMX(550) 1605 D18  ; 自动运行条件延时时间
; rung 5
LD P_On
AND H81.02  ; 提速度
ANDNOT H31.08  ; 1#模组抽真空
ANDNOT H33.08  ; 3#模组抽真空
ANDNOT H34.08  ; 4#模组抽真空
TIMX(550) 1691 &10  ; 除#2其他都关闭延时

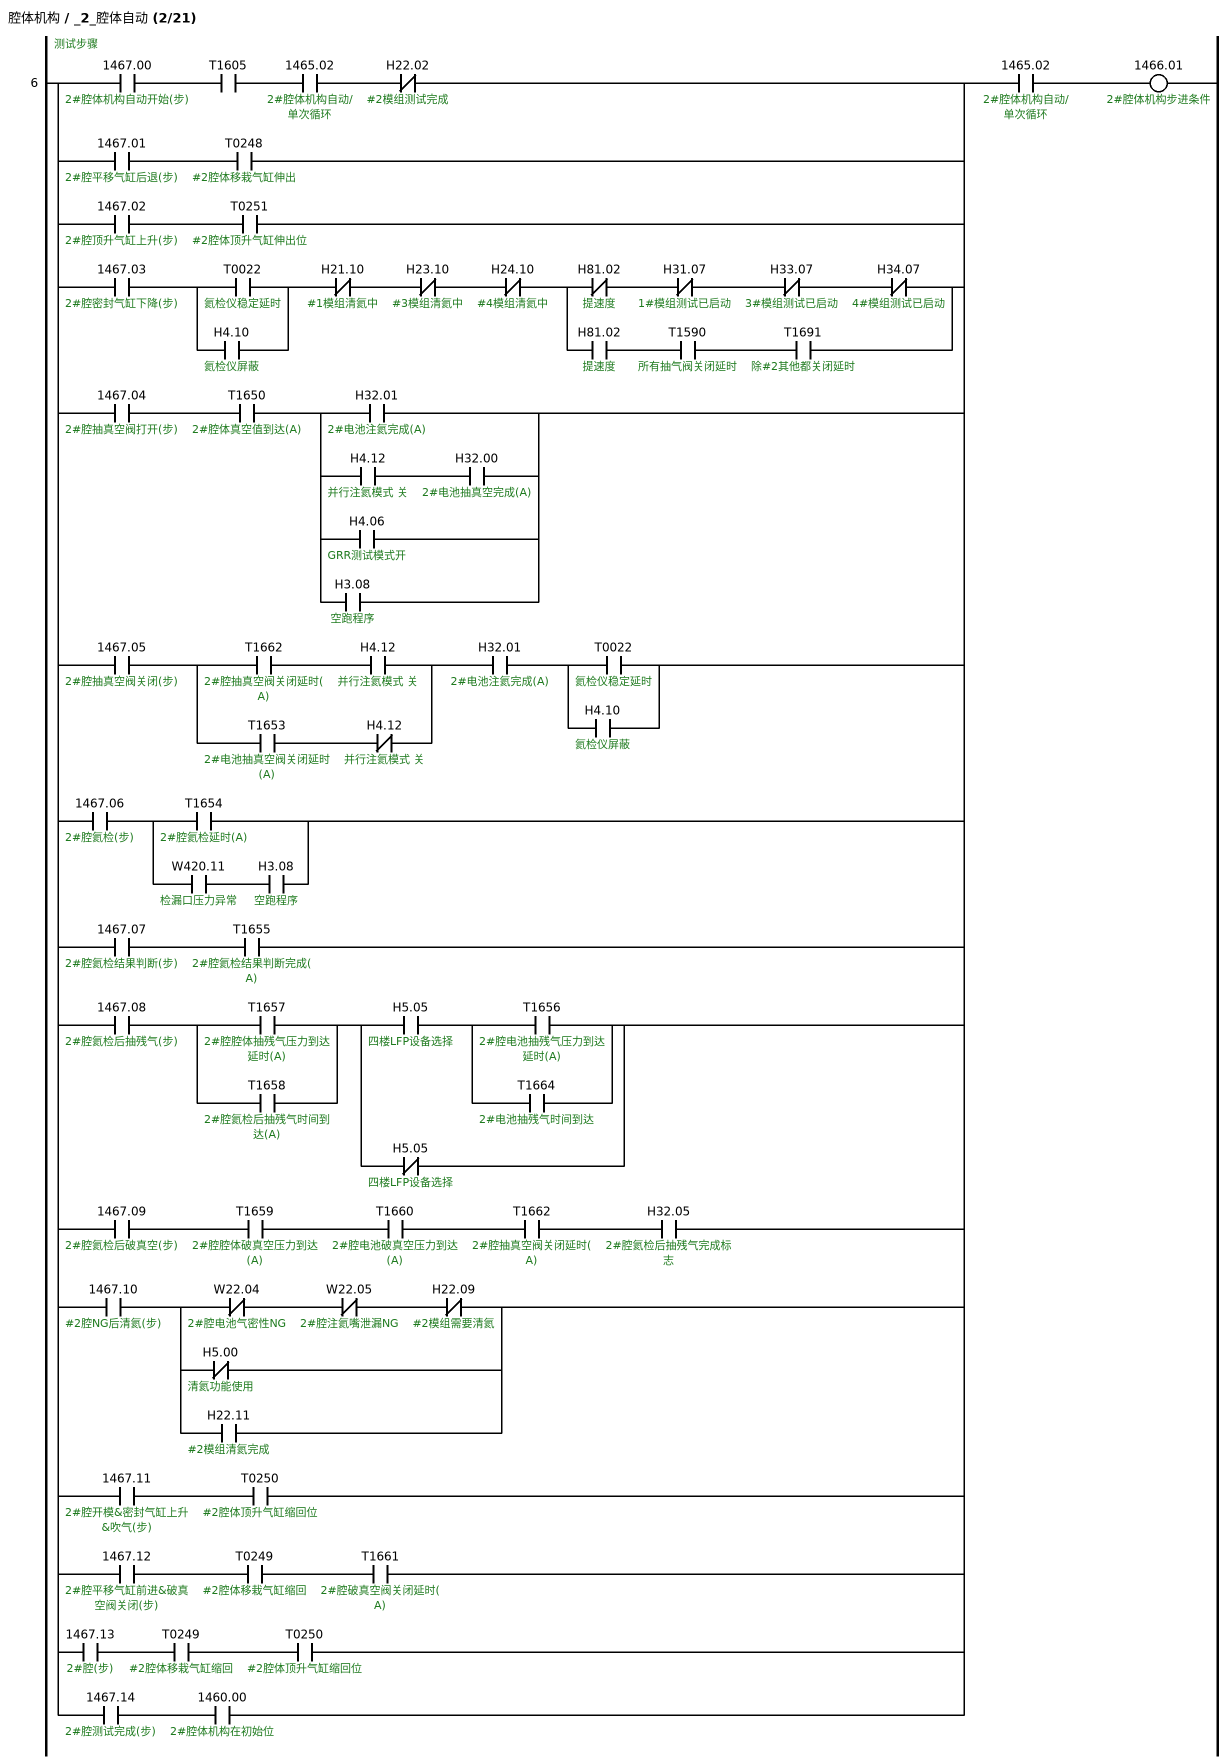
; rung 6: 测试步骤
LD 1467.00  ; 2#腔体机构自动开始(步)
AND T1605
AND 1465.02  ; 2#腔体机构自动/单次循环
ANDNOT H22.02  ; #2模组测试完成
LD 1467.01  ; 2#腔平移气缸后退(步)
AND T0248  ; #2腔体移栽气缸伸出
ORLD
LD 1467.02  ; 2#腔顶升气缸上升(步)
AND T0251  ; #2腔体顶升气缸伸出位
ORLD
LD 1467.03  ; 2#腔密封气缸下降(步)
LD T0022  ; 氦检仪稳定延时
OR H4.10  ; 氦检仪屏蔽
ANDLD
ANDNOT H21.10  ; #1模组清氦中
ANDNOT H23.10  ; #3模组清氦中
ANDNOT H24.10  ; #4模组清氦中
LDNOT H81.02  ; 提速度
ANDNOT H31.07  ; 1#模组测试已启动
ANDNOT H33.07  ; 3#模组测试已启动
ANDNOT H34.07  ; 4#模组测试已启动
LD H81.02  ; 提速度
AND T1590  ; 所有抽气阀关闭延时
AND T1691  ; 除#2其他都关闭延时
ORLD
ANDLD
ORLD
LD 1467.04  ; 2#腔抽真空阀打开(步)
AND T1650  ; 2#腔体真空值到达(A)
LD H32.01  ; 2#电池注氦完成(A)
LD H4.12  ; 并行注氦模式 关
AND H32.00  ; 2#电池抽真空完成(A)
ORLD
OR H4.06  ; GRR测试模式开
OR H3.08  ; 空跑程序
ANDLD
ORLD
LD 1467.05  ; 2#腔抽真空阀关闭(步)
LD T1662  ; 2#腔抽真空阀关闭延时(A)
AND H4.12  ; 并行注氦模式 关
LD T1653  ; 2#电池抽真空阀关闭延时(A)
ANDNOT H4.12  ; 并行注氦模式 关
ORLD
ANDLD
AND H32.01  ; 2#电池注氦完成(A)
LD T0022  ; 氦检仪稳定延时
OR H4.10  ; 氦检仪屏蔽
ANDLD
ORLD
LD 1467.06  ; 2#腔氦检(步)
LD T1654  ; 2#腔氦检延时(A)
LD W420.11  ; 检漏口压力异常
AND H3.08  ; 空跑程序
ORLD
ANDLD
ORLD
LD 1467.07  ; 2#腔氦检结果判断(步)
AND T1655  ; 2#腔氦检结果判断完成(A)
ORLD
LD 1467.08  ; 2#腔氦检后抽残气(步)
LD T1657  ; 2#腔腔体抽残气压力到达延时(A)
OR T1658  ; 2#腔氦检后抽残气时间到达(A)
ANDLD
LD H5.05  ; 四楼LFP设备选择
LD T1656  ; 2#腔电池抽残气压力到达延时(A)
OR T1664  ; 2#电池抽残气时间到达
ANDLD
ORNOT H5.05  ; 四楼LFP设备选择
ANDLD
ORLD
LD 1467.09  ; 2#腔氦检后破真空(步)
AND T1659  ; 2#腔腔体破真空压力到达(A)
AND T1660  ; 2#腔电池破真空压力到达(A)
AND T1662  ; 2#腔抽真空阀关闭延时(A)
AND H32.05  ; 2#腔氦检后抽残气完成标志
ORLD
LD 1467.10  ; #2腔NG后清氦(步)
LDNOT W22.04  ; 2#腔电池气密性NG
ANDNOT W22.05  ; 2#腔注氦嘴泄漏NG
ANDNOT H22.09  ; #2模组需要清氦
ORNOT H5.00  ; 清氦功能使用
OR H22.11  ; #2模组清氦完成
ANDLD
ORLD
LD 1467.11  ; 2#腔开模&密封气缸上升&吹气(步)
AND T0250  ; #2腔体顶升气缸缩回位
ORLD
LD 1467.12  ; 2#腔平移气缸前进&破真空阀关闭(步)
AND T0249  ; #2腔体移栽气缸缩回
AND T1661  ; 2#腔破真空阀关闭延时(A)
ORLD
LD 1467.13  ; 2#腔(步)
AND T0249  ; #2腔体移栽气缸缩回
AND T0250  ; #2腔体顶升气缸缩回位
ORLD
LD 1467.14  ; 2#腔测试完成(步)
AND 1460.00  ; 2#腔体机构在初始位
ORLD
AND 1465.02  ; 2#腔体机构自动/单次循环
OUT 1466.01  ; 2#腔体机构步进条件

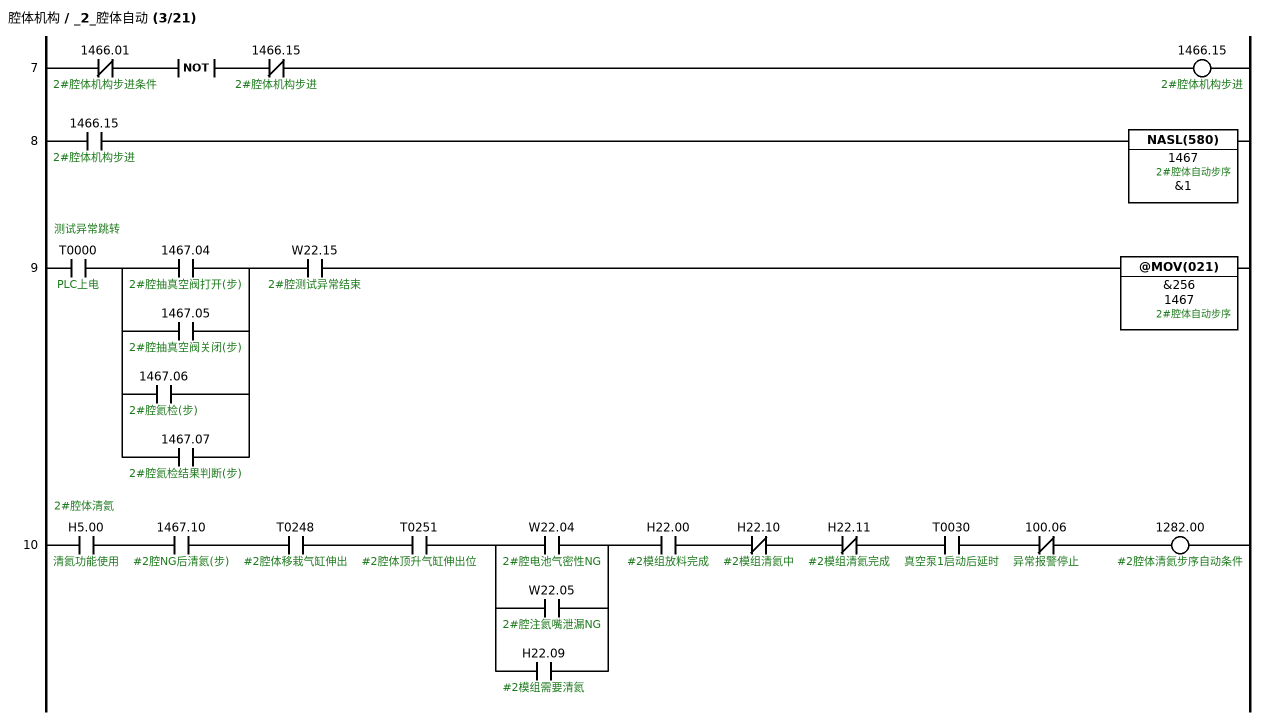
; rung 7
LDNOT 1466.01  ; 2#腔体机构步进条件
NOT(520)
ANDNOT 1466.15  ; 2#腔体机构步进
OUT 1466.15  ; 2#腔体机构步进
; rung 8
LD 1466.15  ; 2#腔体机构步进
NASL(580) 1467 &1  ; 2#腔体自动步序
; rung 9: 测试异常跳转
LD T0000  ; PLC上电
LD 1467.04  ; 2#腔抽真空阀打开(步)
OR 1467.05  ; 2#腔抽真空阀关闭(步)
OR 1467.06  ; 2#腔氦检(步)
OR 1467.07  ; 2#腔氦检结果判断(步)
ANDLD
AND W22.15  ; 2#腔测试异常结束
@MOV(021) &256 1467  ; 2#腔体自动步序
; rung 10: 2#腔体清氦
LD H5.00  ; 清氦功能使用
AND 1467.10  ; #2腔NG后清氦(步)
AND T0248  ; #2腔体移栽气缸伸出
AND T0251  ; #2腔体顶升气缸伸出位
LD W22.04  ; 2#腔电池气密性NG
OR W22.05  ; 2#腔注氦嘴泄漏NG
OR H22.09  ; #2模组需要清氦
ANDLD
AND H22.00  ; #2模组放料完成
ANDNOT H22.10  ; #2模组清氦中
ANDNOT H22.11  ; #2模组清氦完成
AND T0030  ; 真空泵1启动后延时
ANDNOT 100.06  ; 异常报警停止
OUT 1282.00  ; #2腔体清氦步序自动条件

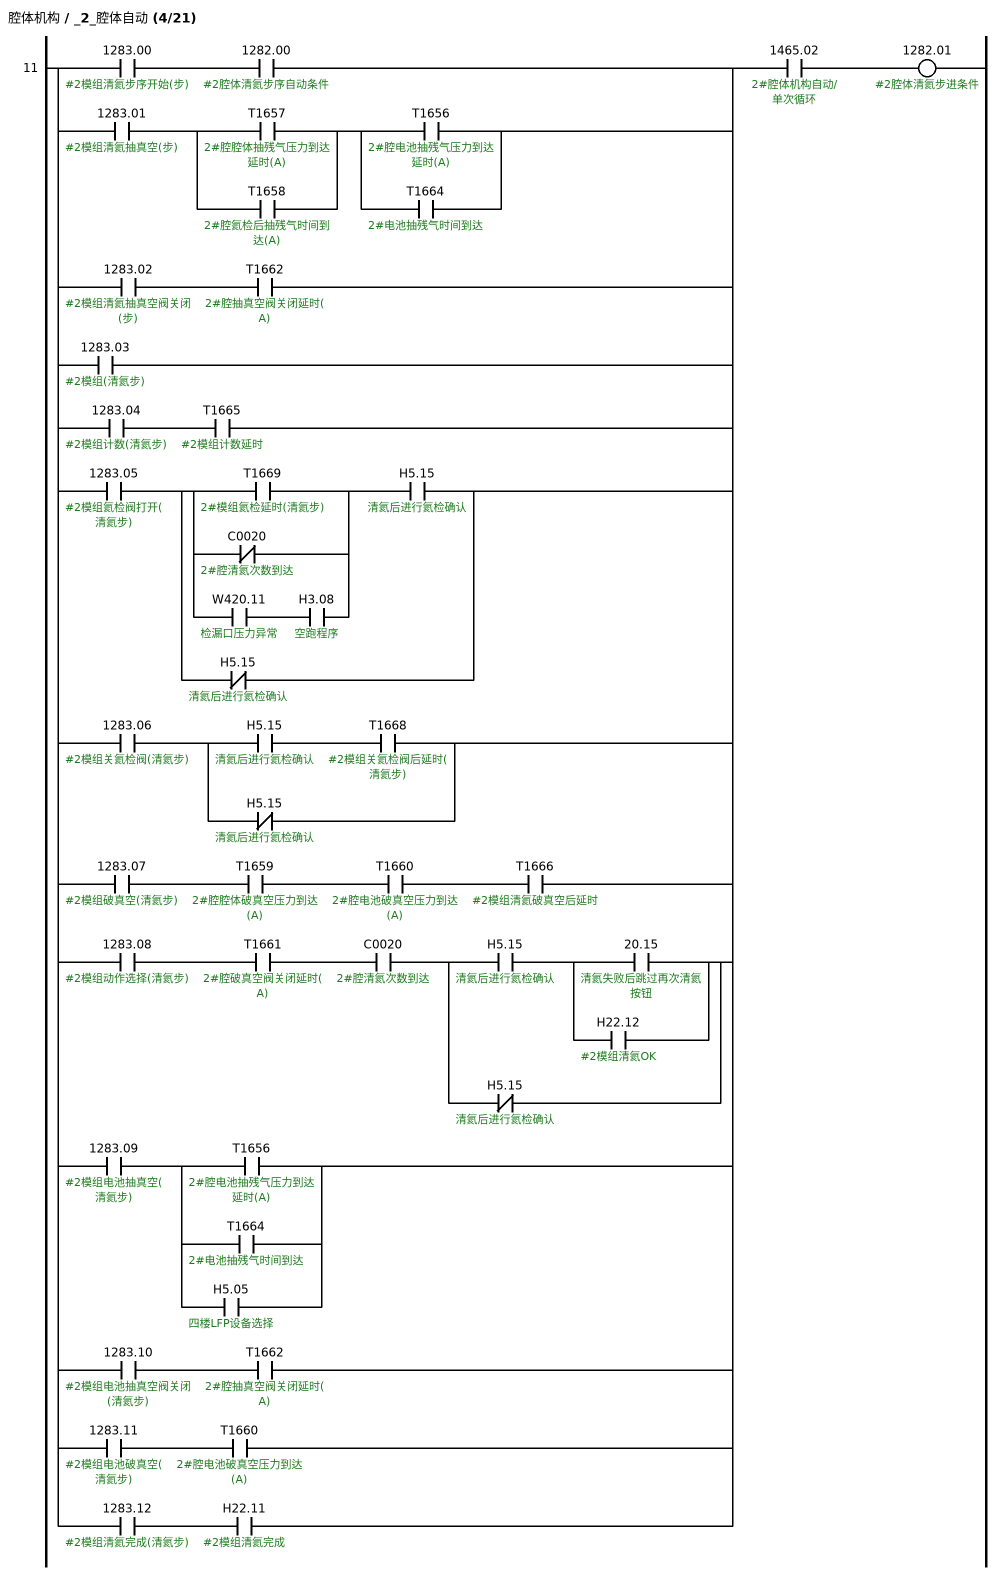
; rung 11
LD 1283.00  ; #2模组清氦步序开始(步)
AND 1282.00  ; #2腔体清氦步序自动条件
LD 1283.01  ; #2模组清氦抽真空(步)
LD T1657  ; 2#腔腔体抽残气压力到达延时(A)
OR T1658  ; 2#腔氦检后抽残气时间到达(A)
ANDLD
LD T1656  ; 2#腔电池抽残气压力到达延时(A)
OR T1664  ; 2#电池抽残气时间到达
ANDLD
ORLD
LD 1283.02  ; #2模组清氦抽真空阀关闭(步)
AND T1662  ; 2#腔抽真空阀关闭延时(A)
ORLD
OR 1283.03  ; #2模组(清氦步)
LD 1283.04  ; #2模组计数(清氦步)
AND T1665  ; #2模组计数延时
ORLD
LD 1283.05  ; #2模组氦检阀打开(清氦步)
LD T1669  ; 2#模组氦检延时(清氦步)
ORNOT C0020  ; 2#腔清氦次数到达
LD W420.11  ; 检漏口压力异常
AND H3.08  ; 空跑程序
ORLD
AND H5.15  ; 清氦后进行氦检确认
ORNOT H5.15  ; 清氦后进行氦检确认
ANDLD
ORLD
LD 1283.06  ; #2模组关氦检阀(清氦步)
LD H5.15  ; 清氦后进行氦检确认
AND T1668  ; #2模组关氦检阀后延时(清氦步)
ORNOT H5.15  ; 清氦后进行氦检确认
ANDLD
ORLD
LD 1283.07  ; #2模组破真空(清氦步)
AND T1659  ; 2#腔腔体破真空压力到达(A)
AND T1660  ; 2#腔电池破真空压力到达(A)
AND T1666  ; #2模组清氦破真空后延时
ORLD
LD 1283.08  ; #2模组动作选择(清氦步)
AND T1661  ; 2#腔破真空阀关闭延时(A)
AND C0020  ; 2#腔清氦次数到达
LD H5.15  ; 清氦后进行氦检确认
LD 20.15  ; 清氦失败后跳过再次清氦按钮
OR H22.12  ; #2模组清氦OK
ANDLD
ORNOT H5.15  ; 清氦后进行氦检确认
ANDLD
ORLD
LD 1283.09  ; #2模组电池抽真空(清氦步)
LD T1656  ; 2#腔电池抽残气压力到达延时(A)
OR T1664  ; 2#电池抽残气时间到达
OR H5.05  ; 四楼LFP设备选择
ANDLD
ORLD
LD 1283.10  ; #2模组电池抽真空阀关闭(清氦步)
AND T1662  ; 2#腔抽真空阀关闭延时(A)
ORLD
LD 1283.11  ; #2模组电池破真空(清氦步)
AND T1660  ; 2#腔电池破真空压力到达(A)
ORLD
LD 1283.12  ; #2模组清氦完成(清氦步)
AND H22.11  ; #2模组清氦完成
ORLD
AND 1465.02  ; 2#腔体机构自动/单次循环
OUT 1282.01  ; #2腔体清氦步进条件

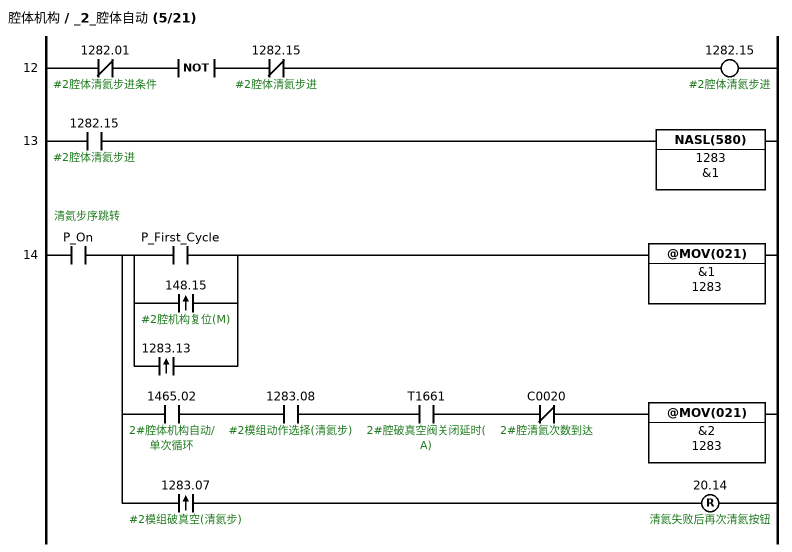
; rung 12
LDNOT 1282.01  ; #2腔体清氦步进条件
NOT(520)
ANDNOT 1282.15  ; #2腔体清氦步进
OUT 1282.15  ; #2腔体清氦步进
; rung 13
LD 1282.15  ; #2腔体清氦步进
NASL(580) 1283 &1
; rung 14: 清氦步序跳转
LD P_On
OUT TR0
LD P_First_Cycle
@OR 148.15  ; #2腔机构复位(M)
@OR 1283.13
ANDLD
@MOV(021) &1 1283
LD TR0
AND 1465.02  ; 2#腔体机构自动/单次循环
AND 1283.08  ; #2模组动作选择(清氦步)
AND T1661  ; 2#腔破真空阀关闭延时(A)
ANDNOT C0020  ; 2#腔清氦次数到达
@MOV(021) &2 1283
LD TR0
@AND 1283.07  ; #2模组破真空(清氦步)
RSET 20.14  ; 清氦失败后再次清氦按钮

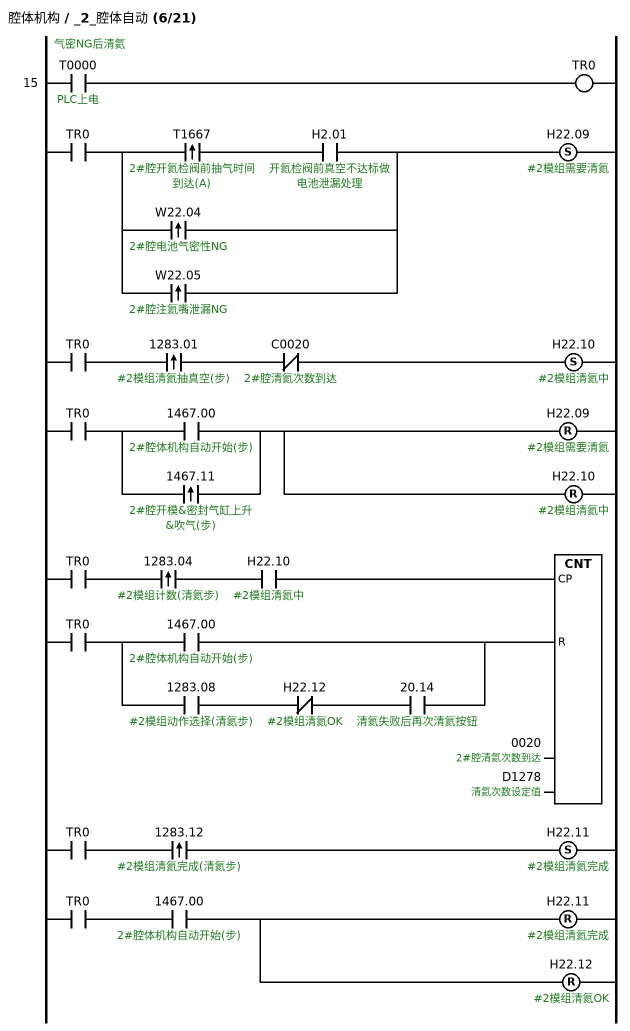
; rung 15: 气密NG后清氦
LD T0000  ; PLC上电
OUT TR0
@LD T1667  ; 2#腔开氦检阀前抽气时间到达(A)
AND H2.01  ; 开氦检阀前真空不达标做电池泄漏处理
@OR W22.04  ; 2#腔电池气密性NG
@OR W22.05  ; 2#腔注氦嘴泄漏NG
ANDLD
SET H22.09  ; #2模组需要清氦
LD TR0
@AND 1283.01  ; #2模组清氦抽真空(步)
ANDNOT C0020  ; 2#腔清氦次数到达
SET H22.10  ; #2模组清氦中
LD TR0
LD 1467.00  ; 2#腔体机构自动开始(步)
@OR 1467.11  ; 2#腔开模&密封气缸上升&吹气(步)
ANDLD
RSET H22.09  ; #2模组需要清氦
RSET H22.10  ; #2模组清氦中
LD TR0
@AND 1283.04  ; #2模组计数(清氦步)
AND H22.10  ; #2模组清氦中
LD TR0
LD 1467.00  ; 2#腔体机构自动开始(步)
LD 1283.08  ; #2模组动作选择(清氦步)
ANDNOT H22.12  ; #2模组清氦OK
AND 20.14  ; 清氦失败后再次清氦按钮
ORLD
ANDLD
CNT 0020 D1278  ; 清氦次数设定值, 2#腔清氦次数到达
LD TR0
@AND 1283.12  ; #2模组清氦完成(清氦步)
SET H22.11  ; #2模组清氦完成
LD TR0
AND 1467.00  ; 2#腔体机构自动开始(步)
RSET H22.11  ; #2模组清氦完成
RSET H22.12  ; #2模组清氦OK

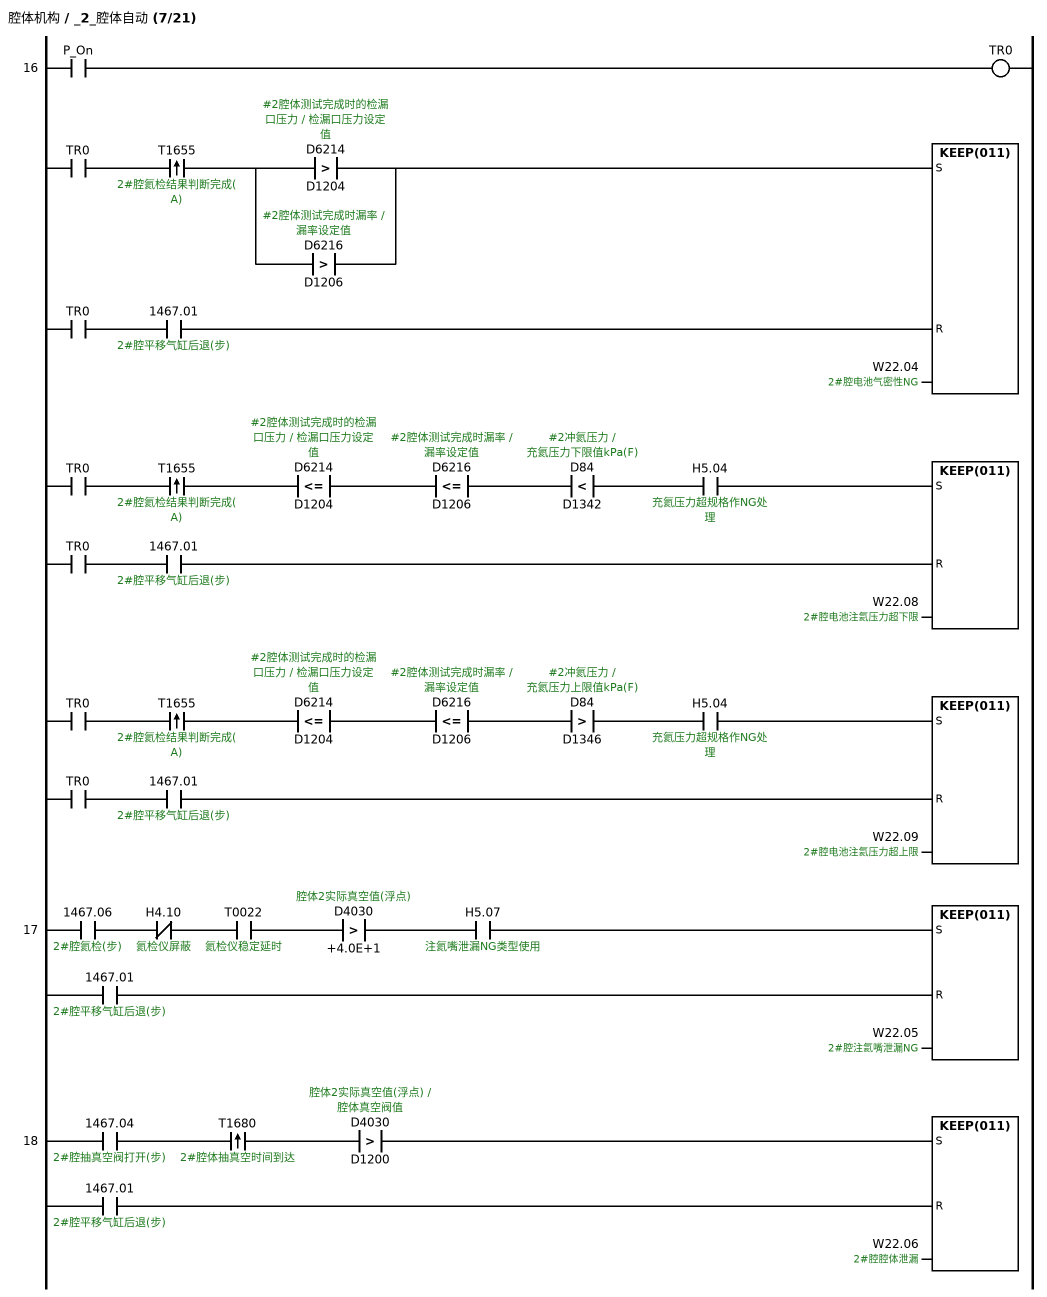
; rung 16
LD P_On
OUT TR0
@AND T1655  ; 2#腔氦检结果判断完成(A)
LD>F(333) D6214 D1204  ; #2腔体测试完成时的检漏口压力, 检漏口压力设定值
OR>F(333) D6216 D1206  ; #2腔体测试完成时漏率, 漏率设定值
ANDLD
LD TR0
AND 1467.01  ; 2#腔平移气缸后退(步)
KEEP(011) W22.04  ; 2#腔电池气密性NG
LD TR0
@AND T1655  ; 2#腔氦检结果判断完成(A)
AND<=F(332) D6214 D1204  ; #2腔体测试完成时的检漏口压力, 检漏口压力设定值
AND<=F(332) D6216 D1206  ; #2腔体测试完成时漏率, 漏率设定值
AND<F(331) D84 D1342  ; #2冲氦压力, 充氦压力下限值kPa(F)
AND H5.04  ; 充氦压力超规格作NG处理
LD TR0
AND 1467.01  ; 2#腔平移气缸后退(步)
KEEP(011) W22.08  ; 2#腔电池注氦压力超下限
LD TR0
@AND T1655  ; 2#腔氦检结果判断完成(A)
AND<=F(332) D6214 D1204  ; #2腔体测试完成时的检漏口压力, 检漏口压力设定值
AND<=F(332) D6216 D1206  ; #2腔体测试完成时漏率, 漏率设定值
AND>F(333) D84 D1346  ; #2冲氦压力, 充氦压力上限值kPa(F)
AND H5.04  ; 充氦压力超规格作NG处理
LD TR0
AND 1467.01  ; 2#腔平移气缸后退(步)
KEEP(011) W22.09  ; 2#腔电池注氦压力超上限
; rung 17
LD 1467.06  ; 2#腔氦检(步)
ANDNOT H4.10  ; 氦检仪屏蔽
AND T0022  ; 氦检仪稳定延时
AND>F(333) D4030 +4.0E+1  ; 腔体2实际真空值(浮点)
AND H5.07  ; 注氦嘴泄漏NG类型使用
LD 1467.01  ; 2#腔平移气缸后退(步)
KEEP(011) W22.05  ; 2#腔注氦嘴泄漏NG
; rung 18
LD 1467.04  ; 2#腔抽真空阀打开(步)
@AND T1680  ; 2#腔体抽真空时间到达
AND>F(333) D4030 D1200  ; 腔体2实际真空值(浮点), 腔体真空阀值
LD 1467.01  ; 2#腔平移气缸后退(步)
KEEP(011) W22.06  ; 2#腔腔体泄漏

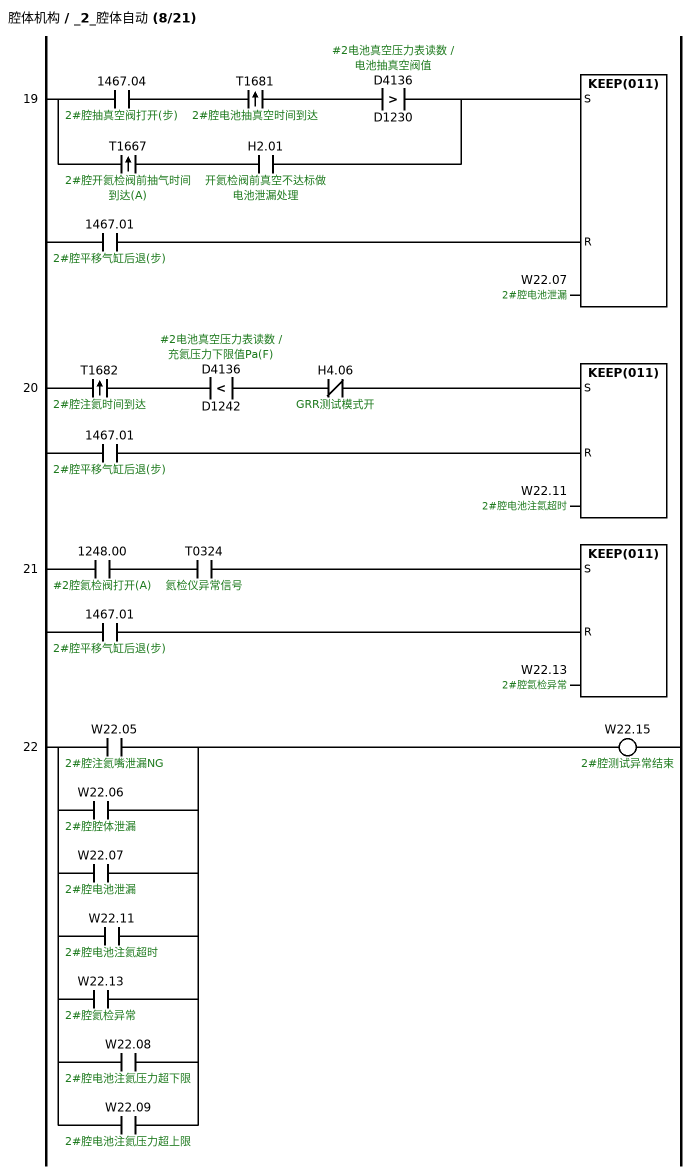
; rung 19
LD 1467.04  ; 2#腔抽真空阀打开(步)
@AND T1681  ; 2#腔电池抽真空时间到达
AND>F(333) D4136 D1230  ; #2电池真空压力表读数, 电池抽真空阀值
@LD T1667  ; 2#腔开氦检阀前抽气时间到达(A)
AND H2.01  ; 开氦检阀前真空不达标做电池泄漏处理
ORLD
LD 1467.01  ; 2#腔平移气缸后退(步)
KEEP(011) W22.07  ; 2#腔电池泄漏
; rung 20
@LD T1682  ; 2#腔注氦时间到达
AND<F(331) D4136 D1242  ; #2电池真空压力表读数, 充氦压力下限值Pa(F)
ANDNOT H4.06  ; GRR测试模式开
LD 1467.01  ; 2#腔平移气缸后退(步)
KEEP(011) W22.11  ; 2#腔电池注氦超时
; rung 21
LD 1248.00  ; #2腔氦检阀打开(A)
AND T0324  ; 氦检仪异常信号
LD 1467.01  ; 2#腔平移气缸后退(步)
KEEP(011) W22.13  ; 2#腔氦检异常
; rung 22
LD W22.05  ; 2#腔注氦嘴泄漏NG
OR W22.06  ; 2#腔腔体泄漏
OR W22.07  ; 2#腔电池泄漏
OR W22.11  ; 2#腔电池注氦超时
OR W22.13  ; 2#腔氦检异常
OR W22.08  ; 2#腔电池注氦压力超下限
OR W22.09  ; 2#腔电池注氦压力超上限
OUT W22.15  ; 2#腔测试异常结束

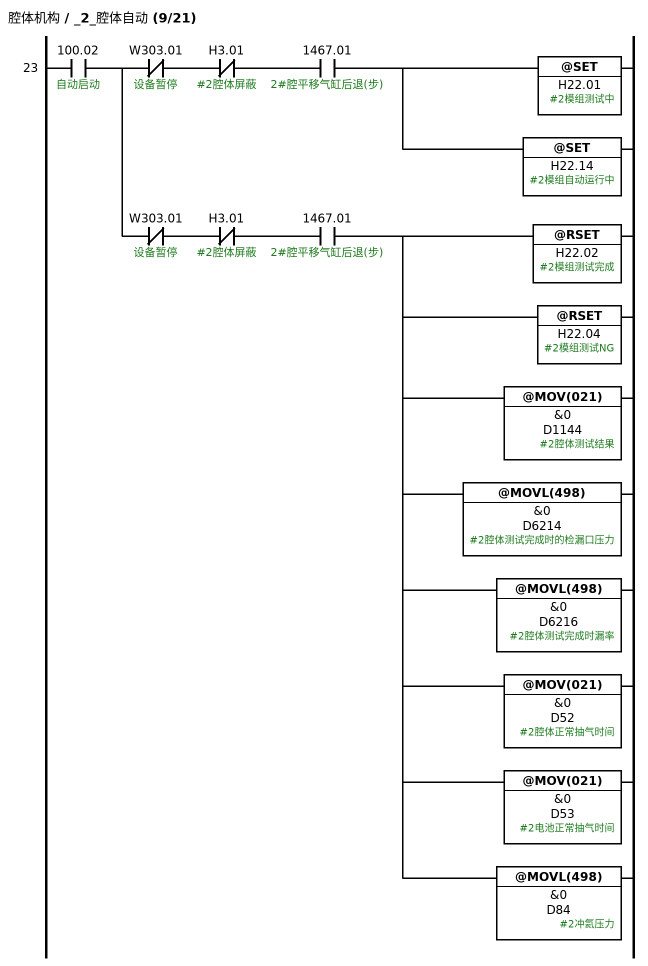
; rung 23
LD 100.02  ; 自动启动
OUT TR0
ANDNOT W303.01  ; 设备暂停
ANDNOT H3.01  ; #2腔体屏蔽
AND 1467.01  ; 2#腔平移气缸后退(步)
@SET H22.01  ; #2模组测试中
@SET H22.14  ; #2模组自动运行中
LD TR0
ANDNOT W303.01  ; 设备暂停
ANDNOT H3.01  ; #2腔体屏蔽
AND 1467.01  ; 2#腔平移气缸后退(步)
@RSET H22.02  ; #2模组测试完成
@RSET H22.04  ; #2模组测试NG
@MOV(021) &0 D1144  ; #2腔体测试结果
@MOVL(498) &0 D6214  ; #2腔体测试完成时的检漏口压力
@MOVL(498) &0 D6216  ; #2腔体测试完成时漏率
@MOV(021) &0 D52  ; #2腔体正常抽气时间
@MOV(021) &0 D53  ; #2电池正常抽气时间
@MOVL(498) &0 D84  ; #2冲氦压力

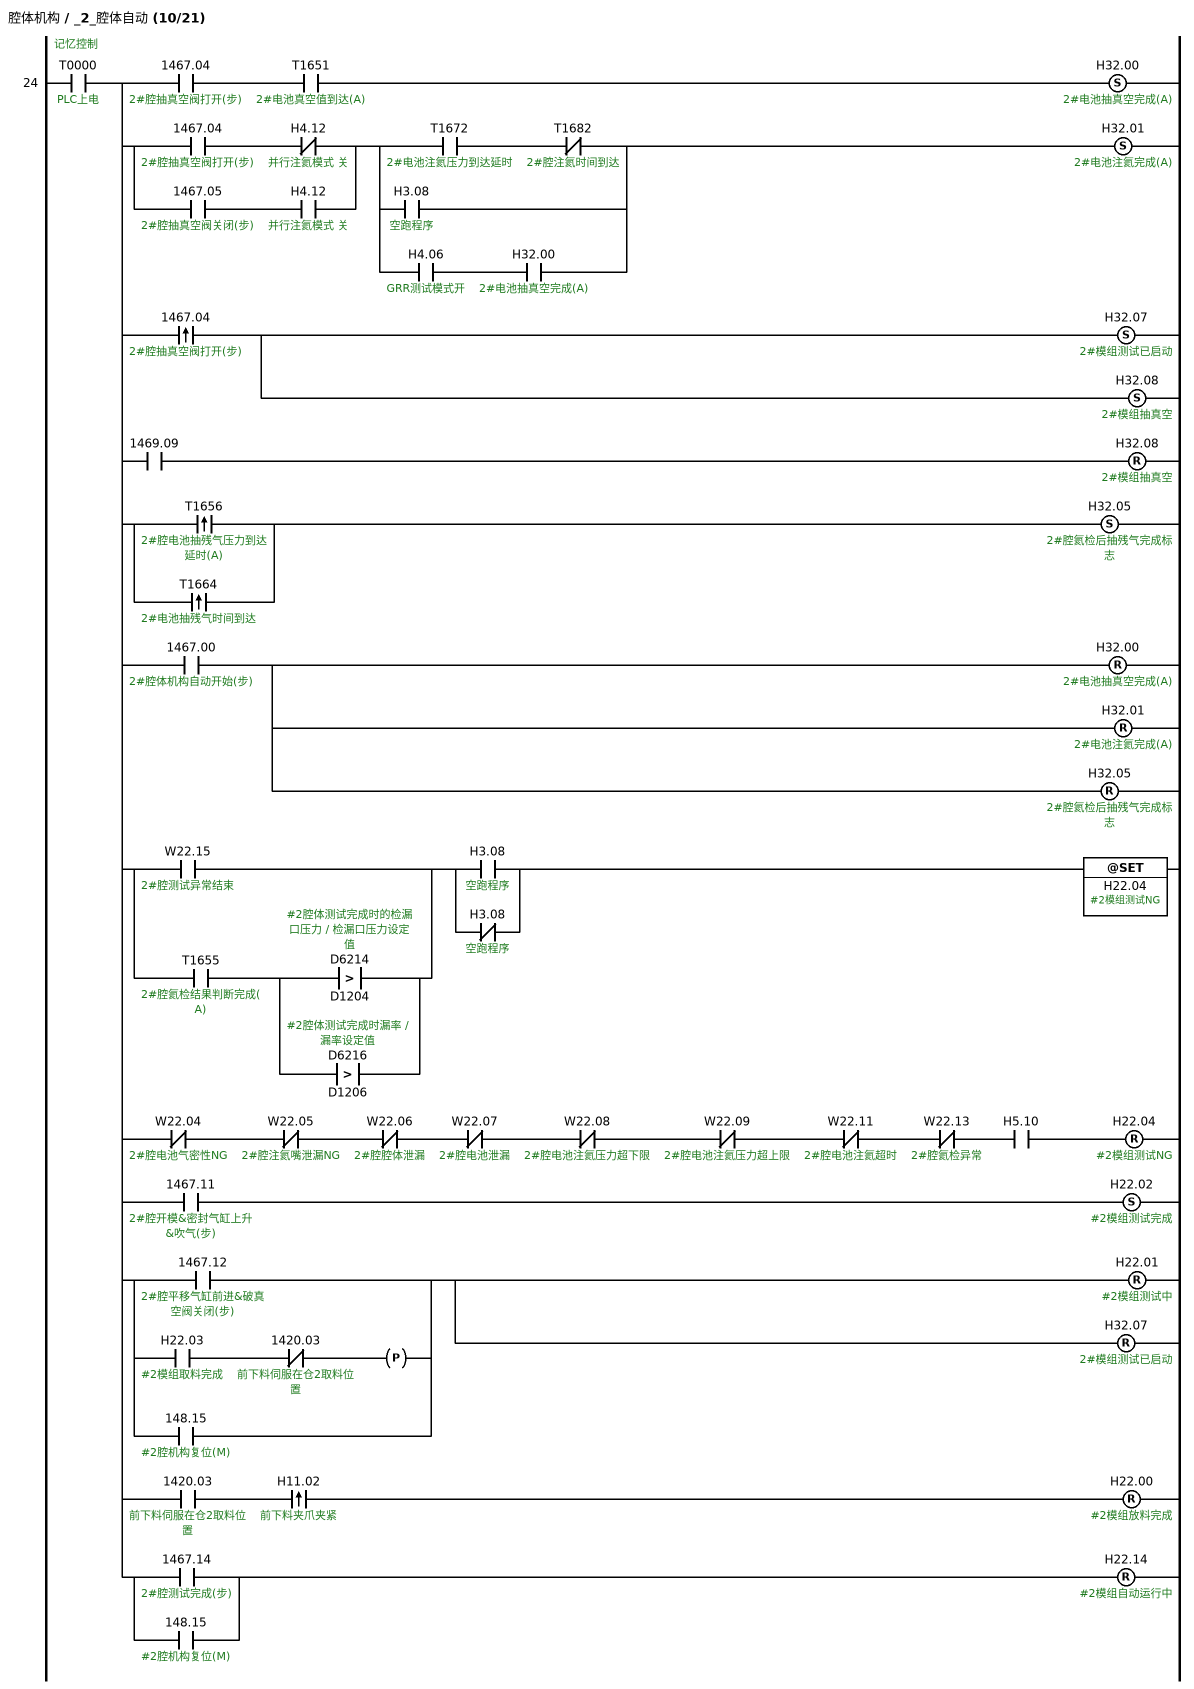
; rung 24: 记忆控制
LD T0000  ; PLC上电
OUT TR0
AND 1467.04  ; 2#腔抽真空阀打开(步)
AND T1651  ; 2#电池真空值到达(A)
SET H32.00  ; 2#电池抽真空完成(A)
LD TR0
LD 1467.04  ; 2#腔抽真空阀打开(步)
ANDNOT H4.12  ; 并行注氦模式 关
LD 1467.05  ; 2#腔抽真空阀关闭(步)
AND H4.12  ; 并行注氦模式 关
ORLD
ANDLD
LD T1672  ; 2#电池注氦压力到达延时
ANDNOT T1682  ; 2#腔注氦时间到达
OR H3.08  ; 空跑程序
LD H4.06  ; GRR测试模式开
AND H32.00  ; 2#电池抽真空完成(A)
ORLD
ANDLD
SET H32.01  ; 2#电池注氦完成(A)
LD TR0
@AND 1467.04  ; 2#腔抽真空阀打开(步)
SET H32.07  ; 2#模组测试已启动
SET H32.08  ; 2#模组抽真空
LD TR0
AND 1469.09
RSET H32.08  ; 2#模组抽真空
LD TR0
@LD T1656  ; 2#腔电池抽残气压力到达延时(A)
@OR T1664  ; 2#电池抽残气时间到达
ANDLD
SET H32.05  ; 2#腔氦检后抽残气完成标志
LD TR0
AND 1467.00  ; 2#腔体机构自动开始(步)
RSET H32.00  ; 2#电池抽真空完成(A)
RSET H32.01  ; 2#电池注氦完成(A)
RSET H32.05  ; 2#腔氦检后抽残气完成标志
LD TR0
LD W22.15  ; 2#腔测试异常结束
LD T1655  ; 2#腔氦检结果判断完成(A)
LD>F(333) D6214 D1204  ; #2腔体测试完成时的检漏口压力, 检漏口压力设定值
OR>F(333) D6216 D1206  ; #2腔体测试完成时漏率, 漏率设定值
ANDLD
ORLD
ANDLD
LD H3.08  ; 空跑程序
ORNOT H3.08  ; 空跑程序
ANDLD
@SET H22.04  ; #2模组测试NG
LD TR0
ANDNOT W22.04  ; 2#腔电池气密性NG
ANDNOT W22.05  ; 2#腔注氦嘴泄漏NG
ANDNOT W22.06  ; 2#腔腔体泄漏
ANDNOT W22.07  ; 2#腔电池泄漏
ANDNOT W22.08  ; 2#腔电池注氦压力超下限
ANDNOT W22.09  ; 2#腔电池注氦压力超上限
ANDNOT W22.11  ; 2#腔电池注氦超时
ANDNOT W22.13  ; 2#腔氦检异常
AND H5.10
RSET H22.04  ; #2模组测试NG
LD TR0
AND 1467.11  ; 2#腔开模&密封气缸上升&吹气(步)
SET H22.02  ; #2模组测试完成
LD TR0
LD 1467.12  ; 2#腔平移气缸前进&破真空阀关闭(步)
LD H22.03  ; #2模组取料完成
ANDNOT 1420.03  ; 前下料伺服在仓2取料位置
UP(521)
ORLD
OR 148.15  ; #2腔机构复位(M)
ANDLD
RSET H22.01  ; #2模组测试中
RSET H32.07  ; 2#模组测试已启动
LD TR0
AND 1420.03  ; 前下料伺服在仓2取料位置
@AND H11.02  ; 前下料夹爪夹紧
RSET H22.00  ; #2模组放料完成
LD TR0
LD 1467.14  ; 2#腔测试完成(步)
OR 148.15  ; #2腔机构复位(M)
ANDLD
RSET H22.14  ; #2模组自动运行中

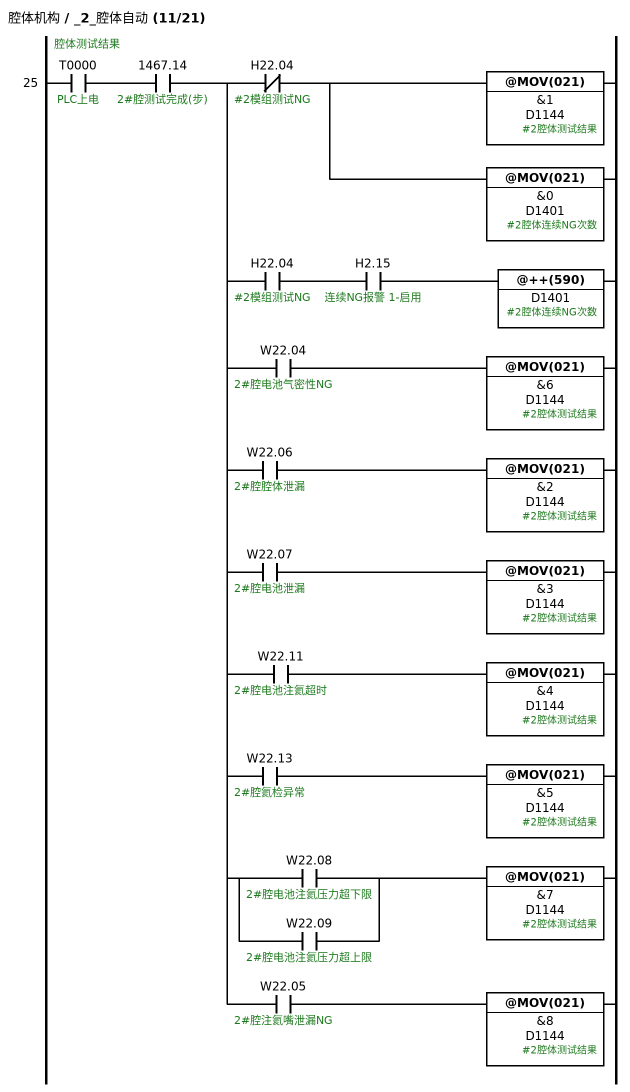
; rung 25: 腔体测试结果
LD T0000  ; PLC上电
AND 1467.14  ; 2#腔测试完成(步)
OUT TR0
ANDNOT H22.04  ; #2模组测试NG
@MOV(021) &1 D1144  ; #2腔体测试结果
@MOV(021) &0 D1401  ; #2腔体连续NG次数
LD TR0
AND H22.04  ; #2模组测试NG
AND H2.15  ; 连续NG报警 1-启用
@++(590) D1401  ; #2腔体连续NG次数
LD TR0
AND W22.04  ; 2#腔电池气密性NG
@MOV(021) &6 D1144  ; #2腔体测试结果
LD TR0
AND W22.06  ; 2#腔腔体泄漏
@MOV(021) &2 D1144  ; #2腔体测试结果
LD TR0
AND W22.07  ; 2#腔电池泄漏
@MOV(021) &3 D1144  ; #2腔体测试结果
LD TR0
AND W22.11  ; 2#腔电池注氦超时
@MOV(021) &4 D1144  ; #2腔体测试结果
LD TR0
AND W22.13  ; 2#腔氦检异常
@MOV(021) &5 D1144  ; #2腔体测试结果
LD TR0
LD W22.08  ; 2#腔电池注氦压力超下限
OR W22.09  ; 2#腔电池注氦压力超上限
ANDLD
@MOV(021) &7 D1144  ; #2腔体测试结果
LD TR0
AND W22.05  ; 2#腔注氦嘴泄漏NG
@MOV(021) &8 D1144  ; #2腔体测试结果

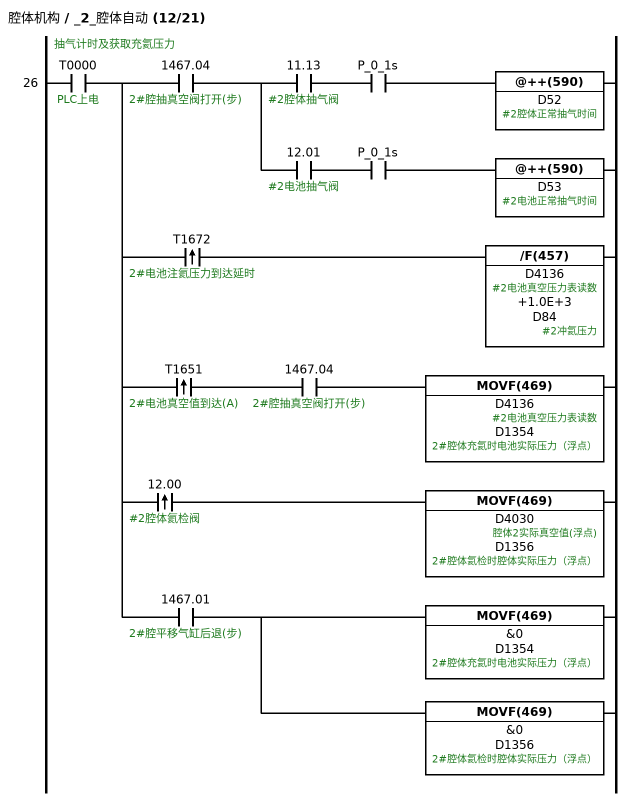
; rung 26: 抽气计时及获取充氦压力
LD T0000  ; PLC上电
OUT TR0
AND 1467.04  ; 2#腔抽真空阀打开(步)
OUT TR1
AND 11.13  ; #2腔体抽气阀
AND P_0_1s
@++(590) D52  ; #2腔体正常抽气时间
LD TR1
AND 12.01  ; #2电池抽气阀
AND P_0_1s
@++(590) D53  ; #2电池正常抽气时间
LD TR0
@AND T1672  ; 2#电池注氦压力到达延时
/F(457) D4136 +1.0E+3 D84  ; #2电池真空压力表读数, #2冲氦压力
LD TR0
@AND T1651  ; 2#电池真空值到达(A)
AND 1467.04  ; 2#腔抽真空阀打开(步)
MOVF(469) D4136 D1354  ; #2电池真空压力表读数, 2#腔体充氦时电池实际压力（浮点）
LD TR0
@AND 12.00  ; #2腔体氦检阀
MOVF(469) D4030 D1356  ; 腔体2实际真空值(浮点), 2#腔体氦检时腔体实际压力（浮点）
LD TR0
AND 1467.01  ; 2#腔平移气缸后退(步)
MOVF(469) &0 D1354  ; 2#腔体充氦时电池实际压力（浮点）
MOVF(469) &0 D1356  ; 2#腔体氦检时腔体实际压力（浮点）

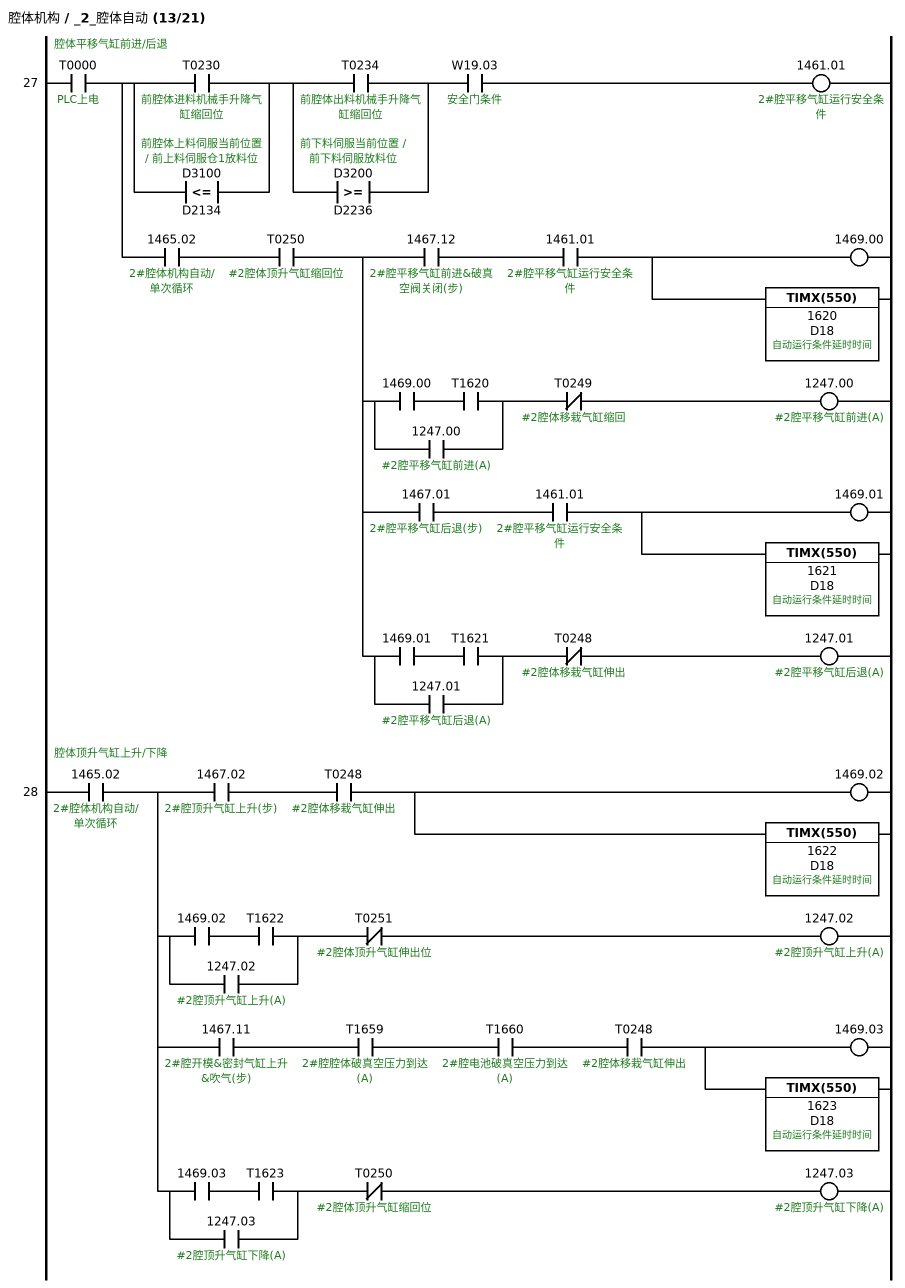
; rung 27: 腔体平移气缸前进/后退
LD T0000  ; PLC上电
OUT TR0
LD T0230  ; 前腔体进料机械手升降气缸缩回位
OR<=SL(318) D3100 D2134  ; 前腔体上料伺服当前位置, 前上料伺服仓1放料位
ANDLD
LD T0234  ; 前腔体出料机械手升降气缸缩回位
OR>=SL(328) D3200 D2236  ; 前下料伺服当前位置, 前下料伺服放料位
ANDLD
AND W19.03  ; 安全门条件
OUT 1461.01  ; 2#腔平移气缸运行安全条件
LD TR0
AND 1465.02  ; 2#腔体机构自动/单次循环
AND T0250  ; #2腔体顶升气缸缩回位
OUT TR0
AND 1467.12  ; 2#腔平移气缸前进&破真空阀关闭(步)
AND 1461.01  ; 2#腔平移气缸运行安全条件
OUT 1469.00
TIMX(550) 1620 D18  ; 自动运行条件延时时间
LD TR0
LD 1469.00
AND T1620
OR 1247.00  ; #2腔平移气缸前进(A)
ANDLD
ANDNOT T0249  ; #2腔体移栽气缸缩回
OUT 1247.00  ; #2腔平移气缸前进(A)
LD TR0
AND 1467.01  ; 2#腔平移气缸后退(步)
AND 1461.01  ; 2#腔平移气缸运行安全条件
OUT 1469.01
TIMX(550) 1621 D18  ; 自动运行条件延时时间
LD TR0
LD 1469.01
AND T1621
OR 1247.01  ; #2腔平移气缸后退(A)
ANDLD
ANDNOT T0248  ; #2腔体移栽气缸伸出
OUT 1247.01  ; #2腔平移气缸后退(A)
; rung 28: 腔体顶升气缸上升/下降
LD 1465.02  ; 2#腔体机构自动/单次循环
OUT TR0
AND 1467.02  ; 2#腔顶升气缸上升(步)
AND T0248  ; #2腔体移栽气缸伸出
OUT 1469.02
TIMX(550) 1622 D18  ; 自动运行条件延时时间
LD TR0
LD 1469.02
AND T1622
OR 1247.02  ; #2腔顶升气缸上升(A)
ANDLD
ANDNOT T0251  ; #2腔体顶升气缸伸出位
OUT 1247.02  ; #2腔顶升气缸上升(A)
LD TR0
AND 1467.11  ; 2#腔开模&密封气缸上升&吹气(步)
AND T1659  ; 2#腔腔体破真空压力到达(A)
AND T1660  ; 2#腔电池破真空压力到达(A)
AND T0248  ; #2腔体移栽气缸伸出
OUT 1469.03
TIMX(550) 1623 D18  ; 自动运行条件延时时间
LD TR0
LD 1469.03
AND T1623
OR 1247.03  ; #2腔顶升气缸下降(A)
ANDLD
ANDNOT T0250  ; #2腔体顶升气缸缩回位
OUT 1247.03  ; #2腔顶升气缸下降(A)

